(* Logix 5000 project; controller reports 1756-L63 rev 20.11; software revision 20.04; part 42 of 52 *)

        [102].log_data[71].valid := 1, [102].log_data[72].valid := 1, [102].log_data[73].valid := 1, [102].log_data[74].valid := 1, [102].log_data[75].valid := 1, [102].log_data[76].valid := 1, [102].log_data[77].valid := 1, [102].log_data[78].valid := 1, [102].log_data[79].valid := 1, [102].log_data[80].valid := 1, [102].log_data[81].valid := 1, [102].log_data[82].valid := 1, [102].log_data[83].valid := 1, [102].log_data[84].valid := 1, [102].log_data[85].valid := 1, [102].log_data[86].valid := 1, [102].log_data[87].valid := 1, [102].log_data[88].valid := 1, [102].log_data[89].valid := 1, [102].log_data[90].valid := 1, [102].log_data[91].valid := 1, [102].log_data[92].valid := 1, [102].log_data[93].valid := 1, [102].log_data[94].valid := 1, [102].log_data[95].valid := 1, [102].log_data[96].valid := 1, [102].log_data[97].valid := 1, [102].log_data[98].valid := 1, [102].log_data[99].valid := 1, [102].log_data[100].valid := 1, [102].log_data[101].valid := 1, [102].log_data[102].valid := 1, [102].log_data[103].valid := 1, [102].log_data[104].valid := 1, [102].log_data[105].valid := 1, [102].log_data[106].valid := 1, [102].log_data[107].valid := 1, [102].log_data[108].valid := 1, [102].log_data[109].valid := 1, [102].log_data[110].valid := 1, [102].log_data[111].valid := 1, [102].log_data[112].valid := 1, [102].log_data[113].valid := 1, [102].log_data[114].valid := 1, [102].log_data[115].valid := 1, [102].log_data[116].valid := 1, [102].log_data[117].valid := 1, [102].log_data[118].valid := 1, [102].log_data[119].valid := 1, [102].log_data[120].valid := 1, [102].log_data[121].valid := 1, [102].log_data[122].valid := 1, [102].log_data[123].valid := 1, [102].log_data[124].valid := 1, [102].time.Year := 2023, [102].time.Month := 1, [102].time.Day := 17, [102].time.Hour := 9, [102].time.Minute := 59, [102].time.Second := 59,
        [103].log_data[0].min := 1.0, [103].log_data[0].max := 1.0, [103].log_data[0].total := 3600.0, [103].log_data[0].time := 3600.0, [103].log_data[0].valid := 1, [103].log_data[1].max := 1.0, [103].log_data[1].total := 558.0, [103].log_data[1].time := 3600.0, [103].log_data[1].maxminute := 47, [103].log_data[1].valid := 1, [103].log_data[2].max := 1.0, [103].log_data[2].total := 554.5, [103].log_data[2].time := 3600.0, [103].log_data[2].maxminute := 47, [103].log_data[2].valid := 1, [103].log_data[3].time := 3600.0, [103].log_data[3].valid := 1, [103].log_data[4].time := 3600.0, [103].log_data[4].valid := 1, [103].log_data[5].max := 1.0, [103].log_data[5].total := 240.0, [103].log_data[5].time := 3600.0, [103].log_data[5].maxminute := 50, [103].log_data[5].valid := 1, [103].log_data[6].time := 3600.0, [103].log_data[6].valid := 1, [103].log_data[7].time := 3600.0, [103].log_data[7].valid := 1, [103].log_data[8].min := 1.0, [103].log_data[8].max := 1.0, [103].log_data[8].total := 3600.0, [103].log_data[8].time := 3600.0, [103].log_data[8].valid := 1, [103].log_data[9].min := 1.0, [103].log_data[9].max := 1.0, [103].log_data[9].total := 3600.0, [103].log_data[9].time := 3600.0, [103].log_data[9].valid := 1, [103].log_data[10].min := 1.0, [103].log_data[10].max := 1.0, [103].log_data[10].total := 3600.0, [103].log_data[10].time := 3600.0, [103].log_data[10].valid := 1, [103].log_data[11].time := 3600.0, [103].log_data[11].valid := 1, [103].log_data[12].min := 1.0, [103].log_data[12].max := 1.0, [103].log_data[12].total := 3600.0, [103].log_data[12].time := 3600.0, [103].log_data[12].valid := 1, [103].log_data[13].min := 1.0, [103].log_data[13].max := 1.0, [103].log_data[13].total := 3600.0, [103].log_data[13].time := 3600.0, [103].log_data[13].valid := 1, [103].log_data[14].time := 3600.0, [103].log_data[14].valid := 1, [103].log_data[15].time := 3600.0, [103].log_data[15].valid := 1, [103].log_data[16].time := 3600.0,
        [103].log_data[16].valid := 1, [103].log_data[17].min := 1.0, [103].log_data[17].max := 1.0, [103].log_data[17].total := 3600.0, [103].log_data[17].time := 3600.0, [103].log_data[17].valid := 1, [103].log_data[18].time := 3600.0, [103].log_data[18].valid := 1, [103].log_data[19].time := 3600.0, [103].log_data[19].valid := 1, [103].log_data[20].time := 3600.0, [103].log_data[20].valid := 1, [103].log_data[21].min := 1.0, [103].log_data[21].max := 1.0, [103].log_data[21].total := 3600.0, [103].log_data[21].time := 3600.0, [103].log_data[21].valid := 1, [103].log_data[22].time := 3600.0, [103].log_data[22].valid := 1, [103].log_data[23].time := 3600.0, [103].log_data[23].valid := 1, [103].log_data[24].time := 3600.0, [103].log_data[24].valid := 1, [103].log_data[25].time := 3600.0, [103].log_data[25].valid := 1, [103].log_data[26].time := 3600.0, [103].log_data[26].valid := 1, [103].log_data[27].time := 3600.0, [103].log_data[27].valid := 1, [103].log_data[28].time := 3600.0, [103].log_data[28].valid := 1, [103].log_data[29].min := 1.0, [103].log_data[29].max := 1.0, [103].log_data[29].total := 3600.0, [103].log_data[29].time := 3600.0, [103].log_data[29].valid := 1, [103].log_data[30].min := 1.0, [103].log_data[30].max := 1.0, [103].log_data[30].total := 3600.0, [103].log_data[30].time := 3600.0, [103].log_data[30].valid := 1, [103].log_data[31].max := 1.0, [103].log_data[31].total := 1440.7471, [103].log_data[31].time := 3600.0, [103].log_data[31].minminute := 3, [103].log_data[31].valid := 1, [103].log_data[32].max := 1.0, [103].log_data[32].total := 1629.7471, [103].log_data[32].time := 3600.0, [103].log_data[32].maxminute := 4, [103].log_data[32].valid := 1, [103].log_data[33].time := 3600.0, [103].log_data[33].valid := 1, [103].log_data[34].time := 3600.0, [103].log_data[34].valid := 1, [103].log_data[35].max := 1.0, [103].log_data[35].total := 1541.7471, [103].log_data[35].time := 3600.0, [103].log_data[35].maxminute := 10, [103].log_data[35].valid := 1,
        [103].log_data[36].max := 1.0, [103].log_data[36].total := 1616.998, [103].log_data[36].time := 3600.0, [103].log_data[36].minminute := 8, [103].log_data[36].valid := 1, [103].log_data[37].max := 7.337698, [103].log_data[37].total := 3557.1064, [103].log_data[37].time := 3600.0, [103].log_data[37].maxminute := 51, [103].log_data[37].valid := 1, [103].log_data[38].time := 3600.0, [103].log_data[38].valid := 1, [103].log_data[39].min := 0.9945885, [103].log_data[39].max := 1.0217944, [103].log_data[39].total := 3607.459, [103].log_data[39].time := 3600.0, [103].log_data[39].minminute := 6, [103].log_data[39].maxminute := 50, [103].log_data[39].valid := 1, [103].log_data[40].min := 7.5945454, [103].log_data[40].max := 7.603614, [103].log_data[40].total := 27364.693, [103].log_data[40].time := 3600.0, [103].log_data[40].minminute := 59, [103].log_data[40].maxminute := 11, [103].log_data[40].valid := 1, [103].log_data[41].min := 0.02273633, [103].log_data[41].max := 0.02411035, [103].log_data[41].total := 82.59197, [103].log_data[41].time := 3600.0, [103].log_data[41].maxminute := 16, [103].log_data[41].valid := 1, [103].log_data[42].min := 2.2916427, [103].log_data[42].max := 2.296236, [103].log_data[42].total := 8258.847, [103].log_data[42].time := 3600.0, [103].log_data[42].minminute := 6, [103].log_data[42].maxminute := 49, [103].log_data[42].valid := 1, [103].log_data[43].min := -0.27999878, [103].log_data[43].max := -0.26000214, [103].log_data[43].total := -993.9634, [103].log_data[43].time := 3600.0, [103].log_data[43].valid := 1, [103].log_data[44].min := -0.3199997, [103].log_data[44].max := -0.30000305, [103].log_data[44].total := -1080.9617, [103].log_data[44].time := 3600.0, [103].log_data[44].minminute := 2, [103].log_data[44].valid := 1, [103].log_data[45].time := 3600.0, [103].log_data[45].valid := 1, [103].log_data[46].time := 3600.0, [103].log_data[46].valid := 1, [103].log_data[47].time := 3600.0, [103].log_data[47].valid := 1, [103].log_data[48].min := 6.732198, [103].log_data[48].max := 6.899556, [103].log_data[48].total := 24363.74, [103].log_data[48].time := 3600.0,
        [103].log_data[48].minminute := 49, [103].log_data[48].maxminute := 53, [103].log_data[48].valid := 1, [103].log_data[49].min := 7.888525, [103].log_data[49].max := 9.465529, [103].log_data[49].total := 32666.957, [103].log_data[49].time := 3600.0, [103].log_data[49].maxminute := 49, [103].log_data[49].valid := 1, [103].log_data[50].min := 1.9457378, [103].log_data[50].max := 2.058684, [103].log_data[50].total := 7166.7627, [103].log_data[50].time := 3600.0, [103].log_data[50].minminute := 50, [103].log_data[50].maxminute := 58, [103].log_data[50].valid := 1, [103].log_data[51].time := 3600.0, [103].log_data[51].valid := 1, [103].log_data[52].min := -3.0800018, [103].log_data[52].max := 0.11999512, [103].log_data[52].total := -7540.314, [103].log_data[52].time := 3600.0, [103].log_data[52].minminute := 9, [103].log_data[52].maxminute := 3, [103].log_data[52].valid := 1, [103].log_data[53].min := -2.8600006, [103].log_data[53].max := 0.2599945, [103].log_data[53].total := -7208.585, [103].log_data[53].time := 3600.0, [103].log_data[53].minminute := 14, [103].log_data[53].maxminute := 30, [103].log_data[53].valid := 1, [103].log_data[54].max := 0.53, [103].log_data[54].total := 1217.2987, [103].log_data[54].time := 3600.0, [103].log_data[54].minminute := 3, [103].log_data[54].maxminute := 25, [103].log_data[54].valid := 1, [103].log_data[55].max := 0.52349997, [103].log_data[55].total := 1254.156, [103].log_data[55].time := 3600.0, [103].log_data[55].minminute := 8, [103].log_data[55].maxminute := 31, [103].log_data[55].valid := 1, [103].log_data[56].min := 0.1594997, [103].log_data[56].max := 0.16012783, [103].log_data[56].total := 575.3569, [103].log_data[56].time := 3600.0, [103].log_data[56].minminute := 39, [103].log_data[56].maxminute := 10, [103].log_data[56].valid := 1, [103].log_data[57].min := 0.23228458, [103].log_data[57].max := 0.23275566, [103].log_data[57].total := 836.9818, [103].log_data[57].time := 3600.0, [103].log_data[57].minminute := 52, [103].log_data[57].maxminute := 25, [103].log_data[57].valid := 1, [103].log_data[58].time := 3600.0, [103].log_data[58].valid := 1,
        [103].log_data[59].time := 3600.0, [103].log_data[59].valid := 1, [103].log_data[60].valid := 1, [103].log_data[61].valid := 1, [103].log_data[62].valid := 1, [103].log_data[63].valid := 1, [103].log_data[64].valid := 1, [103].log_data[65].valid := 1, [103].log_data[66].valid := 1, [103].log_data[67].valid := 1, [103].log_data[68].valid := 1, [103].log_data[69].valid := 1, [103].log_data[70].valid := 1, [103].log_data[71].valid := 1, [103].log_data[72].valid := 1, [103].log_data[73].valid := 1, [103].log_data[74].valid := 1, [103].log_data[75].valid := 1, [103].log_data[76].valid := 1, [103].log_data[77].valid := 1, [103].log_data[78].valid := 1, [103].log_data[79].valid := 1, [103].log_data[80].valid := 1, [103].log_data[81].valid := 1, [103].log_data[82].valid := 1, [103].log_data[83].valid := 1, [103].log_data[84].valid := 1, [103].log_data[85].valid := 1, [103].log_data[86].valid := 1, [103].log_data[87].valid := 1, [103].log_data[88].valid := 1, [103].log_data[89].valid := 1, [103].log_data[90].valid := 1, [103].log_data[91].valid := 1, [103].log_data[92].valid := 1, [103].log_data[93].valid := 1, [103].log_data[94].valid := 1, [103].log_data[95].valid := 1, [103].log_data[96].valid := 1, [103].log_data[97].valid := 1, [103].log_data[98].valid := 1, [103].log_data[99].valid := 1, [103].log_data[100].valid := 1, [103].log_data[101].valid := 1, [103].log_data[102].valid := 1, [103].log_data[103].valid := 1, [103].log_data[104].valid := 1, [103].log_data[105].valid := 1, [103].log_data[106].valid := 1, [103].log_data[107].valid := 1, [103].log_data[108].valid := 1, [103].log_data[109].valid := 1, [103].log_data[110].valid := 1, [103].log_data[111].valid := 1, [103].log_data[112].valid := 1, [103].log_data[113].valid := 1, [103].log_data[114].valid := 1, [103].log_data[115].valid := 1, [103].log_data[116].valid := 1, [103].log_data[117].valid := 1,
        [103].log_data[118].valid := 1, [103].log_data[119].valid := 1, [103].log_data[120].valid := 1, [103].log_data[121].valid := 1, [103].log_data[122].valid := 1, [103].log_data[123].valid := 1, [103].log_data[124].valid := 1, [103].time.Year := 2023, [103].time.Month := 1, [103].time.Day := 17, [103].time.Hour := 10, [103].time.Minute := 59, [103].time.Second := 59, [104].log_data[0].min := 1.0, [104].log_data[0].max := 1.0, [104].log_data[0].total := 3600.0, [104].log_data[0].time := 3600.0, [104].log_data[0].valid := 1, [104].log_data[1].max := 1.0, [104].log_data[1].total := 90.0, [104].log_data[1].time := 3600.0, [104].log_data[1].maxminute := 5, [104].log_data[1].valid := 1, [104].log_data[2].max := 1.0, [104].log_data[2].total := 86.5, [104].log_data[2].time := 3600.0, [104].log_data[2].maxminute := 5, [104].log_data[2].valid := 1, [104].log_data[3].time := 3600.0, [104].log_data[3].valid := 1, [104].log_data[4].time := 3600.0, [104].log_data[4].valid := 1, [104].log_data[5].time := 3600.0, [104].log_data[5].valid := 1, [104].log_data[6].time := 3600.0, [104].log_data[6].valid := 1, [104].log_data[7].time := 3600.0, [104].log_data[7].valid := 1, [104].log_data[8].min := 1.0, [104].log_data[8].max := 1.0, [104].log_data[8].total := 3600.0, [104].log_data[8].time := 3600.0, [104].log_data[8].valid := 1, [104].log_data[9].min := 1.0, [104].log_data[9].max := 1.0, [104].log_data[9].total := 3600.0, [104].log_data[9].time := 3600.0, [104].log_data[9].valid := 1, [104].log_data[10].min := 1.0, [104].log_data[10].max := 1.0, [104].log_data[10].total := 3600.0, [104].log_data[10].time := 3600.0, [104].log_data[10].valid := 1, [104].log_data[11].time := 3600.0, [104].log_data[11].valid := 1, [104].log_data[12].min := 1.0, [104].log_data[12].max := 1.0, [104].log_data[12].total := 3600.0, [104].log_data[12].time := 3600.0, [104].log_data[12].valid := 1,
        [104].log_data[13].min := 1.0, [104].log_data[13].max := 1.0, [104].log_data[13].total := 3600.0, [104].log_data[13].time := 3600.0, [104].log_data[13].valid := 1, [104].log_data[14].time := 3600.0, [104].log_data[14].valid := 1, [104].log_data[15].time := 3600.0, [104].log_data[15].valid := 1, [104].log_data[16].time := 3600.0, [104].log_data[16].valid := 1, [104].log_data[17].min := 1.0, [104].log_data[17].max := 1.0, [104].log_data[17].total := 3600.0, [104].log_data[17].time := 3600.0, [104].log_data[17].valid := 1, [104].log_data[18].time := 3600.0, [104].log_data[18].valid := 1, [104].log_data[19].time := 3600.0, [104].log_data[19].valid := 1, [104].log_data[20].time := 3600.0, [104].log_data[20].valid := 1, [104].log_data[21].min := 1.0, [104].log_data[21].max := 1.0, [104].log_data[21].total := 3600.0, [104].log_data[21].time := 3600.0, [104].log_data[21].valid := 1, [104].log_data[22].time := 3600.0, [104].log_data[22].valid := 1, [104].log_data[23].time := 3600.0, [104].log_data[23].valid := 1, [104].log_data[24].time := 3600.0, [104].log_data[24].valid := 1, [104].log_data[25].time := 3600.0, [104].log_data[25].valid := 1, [104].log_data[26].time := 3600.0, [104].log_data[26].valid := 1, [104].log_data[27].time := 3600.0, [104].log_data[27].valid := 1, [104].log_data[28].time := 3600.0, [104].log_data[28].valid := 1, [104].log_data[29].min := 1.0, [104].log_data[29].max := 1.0, [104].log_data[29].total := 3600.0, [104].log_data[29].time := 3600.0, [104].log_data[29].valid := 1, [104].log_data[30].min := 1.0, [104].log_data[30].max := 1.0, [104].log_data[30].total := 3600.0, [104].log_data[30].time := 3600.0, [104].log_data[30].valid := 1, [104].log_data[31].max := 1.0, [104].log_data[31].total := 1469.498, [104].log_data[31].time := 3600.0, [104].log_data[31].minminute := 6, [104].log_data[31].valid := 1, [104].log_data[32].max := 1.0, [104].log_data[32].total := 1629.998, [104].log_data[32].time := 3600.0, [104].log_data[32].maxminute := 7,
        [104].log_data[32].valid := 1, [104].log_data[33].time := 3600.0, [104].log_data[33].valid := 1, [104].log_data[34].time := 3600.0, [104].log_data[34].valid := 1, [104].log_data[35].max := 1.0, [104].log_data[35].total := 1440.498, [104].log_data[35].time := 3600.0, [104].log_data[35].minminute := 1, [104].log_data[35].valid := 1, [104].log_data[36].max := 1.0, [104].log_data[36].total := 1629.7471, [104].log_data[36].time := 3600.0, [104].log_data[36].maxminute := 2, [104].log_data[36].valid := 1, [104].log_data[37].max := 2.600009, [104].log_data[37].total := 99.13652, [104].log_data[37].time := 3600.0, [104].log_data[37].maxminute := 5, [104].log_data[37].valid := 1, [104].log_data[38].time := 3600.0, [104].log_data[38].valid := 1, [104].log_data[39].min := 0.9957663, [104].log_data[39].max := 1.0073081, [104].log_data[39].total := 3607.94, [104].log_data[39].time := 3600.0, [104].log_data[39].minminute := 4, [104].log_data[39].maxminute := 43, [104].log_data[39].valid := 1, [104].log_data[40].min := 7.5802555, [104].log_data[40].max := 7.6093855, [104].log_data[40].total := 27364.307, [104].log_data[40].time := 3600.0, [104].log_data[40].minminute := 45, [104].log_data[40].maxminute := 48, [104].log_data[40].valid := 1, [104].log_data[41].min := 0.02273633, [104].log_data[41].max := 0.023128908, [104].log_data[41].total := 82.71829, [104].log_data[41].time := 3600.0, [104].log_data[41].valid := 1, [104].log_data[42].min := 2.2911716, [104].log_data[42].max := 2.296118, [104].log_data[42].total := 8258.796, [104].log_data[42].time := 3600.0, [104].log_data[42].minminute := 24, [104].log_data[42].maxminute := 29, [104].log_data[42].valid := 1, [104].log_data[43].min := -0.27999878, [104].log_data[43].max := -0.26000214, [104].log_data[43].total := -1007.0374, [104].log_data[43].time := 3600.0, [104].log_data[43].valid := 1, [104].log_data[44].min := -0.3199997, [104].log_data[44].max := -0.30000305, [104].log_data[44].total := -1100.4613, [104].log_data[44].time := 3600.0, [104].log_data[44].valid := 1, [104].log_data[45].time := 3600.0, [104].log_data[45].valid := 1,
        [104].log_data[46].time := 3600.0, [104].log_data[46].valid := 1, [104].log_data[47].time := 3600.0, [104].log_data[47].valid := 1, [104].log_data[48].min := 6.578031, [104].log_data[48].max := 6.801175, [104].log_data[48].total := 24174.486, [104].log_data[48].time := 3600.0, [104].log_data[48].minminute := 16, [104].log_data[48].maxminute := 33, [104].log_data[48].valid := 1, [104].log_data[49].min := 6.728443, [104].log_data[49].max := 9.348344, [104].log_data[49].total := 28856.195, [104].log_data[49].time := 3600.0, [104].log_data[49].minminute := 18, [104].log_data[49].maxminute := 59, [104].log_data[49].valid := 1, [104].log_data[50].min := 1.9717662, [104].log_data[50].max := 2.0559752, [104].log_data[50].total := 7259.038, [104].log_data[50].time := 3600.0, [104].log_data[50].minminute := 59, [104].log_data[50].maxminute := 1, [104].log_data[50].valid := 1, [104].log_data[51].time := 3600.0, [104].log_data[51].valid := 1, [104].log_data[52].min := -2.880005, [104].log_data[52].max := 0.11999512, [104].log_data[52].total := -7743.9883, [104].log_data[52].time := 3600.0, [104].log_data[52].minminute := 7, [104].log_data[52].maxminute := 6, [104].log_data[52].valid := 1, [104].log_data[53].min := -2.540001, [104].log_data[53].max := 0.2400055, [104].log_data[53].total := -7001.7065, [104].log_data[53].time := 3600.0, [104].log_data[53].minminute := 55, [104].log_data[53].maxminute := 2, [104].log_data[53].valid := 1, [104].log_data[54].max := 0.5215, [104].log_data[54].total := 1230.9836, [104].log_data[54].time := 3600.0, [104].log_data[54].minminute := 6, [104].log_data[54].maxminute := 18, [104].log_data[54].valid := 1, [104].log_data[55].max := 0.52099997, [104].log_data[55].total := 1217.138, [104].log_data[55].time := 3600.0, [104].log_data[55].minminute := 1, [104].log_data[55].maxminute := 55, [104].log_data[55].valid := 1, [104].log_data[56].min := 0.15957822, [104].log_data[56].max := 0.16001005, [104].log_data[56].total := 575.15814, [104].log_data[56].time := 3600.0, [104].log_data[56].minminute := 15, [104].log_data[56].maxminute := 7, [104].log_data[56].valid := 1,
        [104].log_data[57].min := 0.2303609, [104].log_data[57].max := 0.23267715, [104].log_data[57].total := 832.2318, [104].log_data[57].time := 3600.0, [104].log_data[57].minminute := 37, [104].log_data[57].valid := 1, [104].log_data[58].time := 3600.0, [104].log_data[58].valid := 1, [104].log_data[59].time := 3600.0, [104].log_data[59].valid := 1, [104].log_data[60].valid := 1, [104].log_data[61].valid := 1, [104].log_data[62].valid := 1, [104].log_data[63].valid := 1, [104].log_data[64].valid := 1, [104].log_data[65].valid := 1, [104].log_data[66].valid := 1, [104].log_data[67].valid := 1, [104].log_data[68].valid := 1, [104].log_data[69].valid := 1, [104].log_data[70].valid := 1, [104].log_data[71].valid := 1, [104].log_data[72].valid := 1, [104].log_data[73].valid := 1, [104].log_data[74].valid := 1, [104].log_data[75].valid := 1, [104].log_data[76].valid := 1, [104].log_data[77].valid := 1, [104].log_data[78].valid := 1, [104].log_data[79].valid := 1, [104].log_data[80].valid := 1, [104].log_data[81].valid := 1, [104].log_data[82].valid := 1, [104].log_data[83].valid := 1, [104].log_data[84].valid := 1, [104].log_data[85].valid := 1, [104].log_data[86].valid := 1, [104].log_data[87].valid := 1, [104].log_data[88].valid := 1, [104].log_data[89].valid := 1, [104].log_data[90].valid := 1, [104].log_data[91].valid := 1, [104].log_data[92].valid := 1, [104].log_data[93].valid := 1, [104].log_data[94].valid := 1, [104].log_data[95].valid := 1, [104].log_data[96].valid := 1, [104].log_data[97].valid := 1, [104].log_data[98].valid := 1, [104].log_data[99].valid := 1, [104].log_data[100].valid := 1, [104].log_data[101].valid := 1, [104].log_data[102].valid := 1, [104].log_data[103].valid := 1, [104].log_data[104].valid := 1, [104].log_data[105].valid := 1, [104].log_data[106].valid := 1, [104].log_data[107].valid := 1, [104].log_data[108].valid := 1, [104].log_data[109].valid := 1,
        [104].log_data[110].valid := 1, [104].log_data[111].valid := 1, [104].log_data[112].valid := 1, [104].log_data[113].valid := 1, [104].log_data[114].valid := 1, [104].log_data[115].valid := 1, [104].log_data[116].valid := 1, [104].log_data[117].valid := 1, [104].log_data[118].valid := 1, [104].log_data[119].valid := 1, [104].log_data[120].valid := 1, [104].log_data[121].valid := 1, [104].log_data[122].valid := 1, [104].log_data[123].valid := 1, [104].log_data[124].valid := 1, [104].time.Year := 2023, [104].time.Month := 1, [104].time.Day := 17, [104].time.Hour := 11, [104].time.Minute := 59, [104].time.Second := 59, [105].log_data[0].min := 1.0, [105].log_data[0].max := 1.0, [105].log_data[0].total := 3600.0, [105].log_data[0].time := 3600.0, [105].log_data[0].valid := 1, [105].log_data[1].max := 1.0, [105].log_data[1].total := 544.0, [105].log_data[1].time := 3600.0, [105].log_data[1].maxminute := 21, [105].log_data[1].valid := 1, [105].log_data[2].max := 1.0, [105].log_data[2].total := 540.5, [105].log_data[2].time := 3600.0, [105].log_data[2].maxminute := 21, [105].log_data[2].valid := 1, [105].log_data[3].time := 3600.0, [105].log_data[3].valid := 1, [105].log_data[4].time := 3600.0, [105].log_data[4].valid := 1, [105].log_data[5].max := 1.0, [105].log_data[5].total := 245.0, [105].log_data[5].time := 3600.0, [105].log_data[5].maxminute := 23, [105].log_data[5].valid := 1, [105].log_data[6].time := 3600.0, [105].log_data[6].valid := 1, [105].log_data[7].time := 3600.0, [105].log_data[7].valid := 1, [105].log_data[8].min := 1.0, [105].log_data[8].max := 1.0, [105].log_data[8].total := 3600.0, [105].log_data[8].time := 3600.0, [105].log_data[8].valid := 1, [105].log_data[9].min := 1.0, [105].log_data[9].max := 1.0, [105].log_data[9].total := 3600.0, [105].log_data[9].time := 3600.0, [105].log_data[9].valid := 1, [105].log_data[10].min := 1.0,
        [105].log_data[10].max := 1.0, [105].log_data[10].total := 3600.0, [105].log_data[10].time := 3600.0, [105].log_data[10].valid := 1, [105].log_data[11].time := 3600.0, [105].log_data[11].valid := 1, [105].log_data[12].min := 1.0, [105].log_data[12].max := 1.0, [105].log_data[12].total := 3600.0, [105].log_data[12].time := 3600.0, [105].log_data[12].valid := 1, [105].log_data[13].min := 1.0, [105].log_data[13].max := 1.0, [105].log_data[13].total := 3600.0, [105].log_data[13].time := 3600.0, [105].log_data[13].valid := 1, [105].log_data[14].time := 3600.0, [105].log_data[14].valid := 1, [105].log_data[15].time := 3600.0, [105].log_data[15].valid := 1, [105].log_data[16].time := 3600.0, [105].log_data[16].valid := 1, [105].log_data[17].min := 1.0, [105].log_data[17].max := 1.0, [105].log_data[17].total := 3600.0, [105].log_data[17].time := 3600.0, [105].log_data[17].valid := 1, [105].log_data[18].time := 3600.0, [105].log_data[18].valid := 1, [105].log_data[19].time := 3600.0, [105].log_data[19].valid := 1, [105].log_data[20].time := 3600.0, [105].log_data[20].valid := 1, [105].log_data[21].min := 1.0, [105].log_data[21].max := 1.0, [105].log_data[21].total := 3600.0, [105].log_data[21].time := 3600.0, [105].log_data[21].valid := 1, [105].log_data[22].time := 3600.0, [105].log_data[22].valid := 1, [105].log_data[23].time := 3600.0, [105].log_data[23].valid := 1, [105].log_data[24].time := 3600.0, [105].log_data[24].valid := 1, [105].log_data[25].time := 3600.0, [105].log_data[25].valid := 1, [105].log_data[26].time := 3600.0, [105].log_data[26].valid := 1, [105].log_data[27].time := 3600.0, [105].log_data[27].valid := 1, [105].log_data[28].time := 3600.0, [105].log_data[28].valid := 1, [105].log_data[29].min := 1.0, [105].log_data[29].max := 1.0, [105].log_data[29].total := 3600.0, [105].log_data[29].time := 3600.0, [105].log_data[29].valid := 1, [105].log_data[30].min := 1.0, [105].log_data[30].max := 1.0, [105].log_data[30].total := 3600.0,
        [105].log_data[30].time := 3600.0, [105].log_data[30].valid := 1, [105].log_data[31].max := 1.0, [105].log_data[31].total := 1629.998, [105].log_data[31].time := 3600.0, [105].log_data[31].valid := 1, [105].log_data[32].max := 1.0, [105].log_data[32].total := 1500.2471, [105].log_data[32].time := 3600.0, [105].log_data[32].maxminute := 11, [105].log_data[32].valid := 1, [105].log_data[33].time := 3600.0, [105].log_data[33].valid := 1, [105].log_data[34].time := 3600.0, [105].log_data[34].valid := 1, [105].log_data[35].max := 1.0, [105].log_data[35].total := 1440.7471, [105].log_data[35].time := 3600.0, [105].log_data[35].minminute := 4, [105].log_data[35].valid := 1, [105].log_data[36].max := 1.0, [105].log_data[36].total := 1629.998, [105].log_data[36].time := 3600.0, [105].log_data[36].maxminute := 6, [105].log_data[36].valid := 1, [105].log_data[37].max := 7.473924, [105].log_data[37].total := 3521.814, [105].log_data[37].time := 3600.0, [105].log_data[37].maxminute := 23, [105].log_data[37].valid := 1, [105].log_data[38].time := 3600.0, [105].log_data[38].valid := 1, [105].log_data[39].min := 0.9950596, [105].log_data[39].max := 1.0221478, [105].log_data[39].total := 3609.72, [105].log_data[39].time := 3600.0, [105].log_data[39].minminute := 39, [105].log_data[39].maxminute := 28, [105].log_data[39].valid := 1, [105].log_data[40].min := 7.5928965, [105].log_data[40].max := 7.6077366, [105].log_data[40].total := 27365.082, [105].log_data[40].time := 3600.0, [105].log_data[40].minminute := 52, [105].log_data[40].maxminute := 54, [105].log_data[40].valid := 1, [105].log_data[41].min := 0.02273633, [105].log_data[41].max := 0.023325196, [105].log_data[41].total := 82.87387, [105].log_data[41].time := 3600.0, [105].log_data[41].minminute := 3, [105].log_data[41].maxminute := 20, [105].log_data[41].valid := 1, [105].log_data[42].min := 2.2917604, [105].log_data[42].max := 2.2964714, [105].log_data[42].total := 8259.048, [105].log_data[42].time := 3600.0, [105].log_data[42].minminute := 22, [105].log_data[42].maxminute := 4, [105].log_data[42].valid := 1,
        [105].log_data[43].min := -0.27999878, [105].log_data[43].max := -0.26000214, [105].log_data[43].total := -998.42554, [105].log_data[43].time := 3600.0, [105].log_data[43].valid := 1, [105].log_data[44].min := -0.3199997, [105].log_data[44].max := -0.30000305, [105].log_data[44].total := -1085.1592, [105].log_data[44].time := 3600.0, [105].log_data[44].valid := 1, [105].log_data[45].time := 3600.0, [105].log_data[45].valid := 1, [105].log_data[46].time := 3600.0, [105].log_data[46].valid := 1, [105].log_data[47].time := 3600.0, [105].log_data[47].valid := 1, [105].log_data[48].min := 6.5708866, [105].log_data[48].max := 6.909449, [105].log_data[48].total := 24175.59, [105].log_data[48].time := 3600.0, [105].log_data[48].minminute := 52, [105].log_data[48].maxminute := 26, [105].log_data[48].valid := 1, [105].log_data[49].min := 6.671519, [105].log_data[49].max := 9.436871, [105].log_data[49].total := 29516.545, [105].log_data[49].time := 3600.0, [105].log_data[49].minminute := 47, [105].log_data[49].maxminute := 17, [105].log_data[49].valid := 1, [105].log_data[50].min := 1.9406737, [105].log_data[50].max := 2.0525599, [105].log_data[50].total := 7204.415, [105].log_data[50].time := 3600.0, [105].log_data[50].minminute := 23, [105].log_data[50].maxminute := 31, [105].log_data[50].valid := 1, [105].log_data[51].time := 3600.0, [105].log_data[51].valid := 1, [105].log_data[52].min := -2.9400024, [105].log_data[52].max := 0.11999512, [105].log_data[52].total := -7841.4717, [105].log_data[52].time := 3600.0, [105].log_data[52].minminute := 32, [105].log_data[52].valid := 1, [105].log_data[53].min := -2.4800034, [105].log_data[53].max := 0.22000122, [105].log_data[53].total := -7097.0947, [105].log_data[53].time := 3600.0, [105].log_data[53].minminute := 25, [105].log_data[53].maxminute := 37, [105].log_data[53].valid := 1, [105].log_data[54].max := 0.5475, [105].log_data[54].total := 1241.1823, [105].log_data[54].time := 3600.0, [105].log_data[54].maxminute := 11, [105].log_data[54].valid := 1, [105].log_data[55].max := 0.52349997, [105].log_data[55].total := 1217.1405, [105].log_data[55].time := 3600.0,
        [105].log_data[55].minminute := 4, [105].log_data[55].maxminute := 16, [105].log_data[55].valid := 1, [105].log_data[56].min := 0.15957822, [105].log_data[56].max := 0.16001005, [105].log_data[56].total := 575.1107, [105].log_data[56].time := 3600.0, [105].log_data[56].minminute := 42, [105].log_data[56].maxminute := 2, [105].log_data[56].valid := 1, [105].log_data[57].min := 0.22894761, [105].log_data[57].max := 0.23083198, [105].log_data[57].total := 829.5313, [105].log_data[57].time := 3600.0, [105].log_data[57].minminute := 59, [105].log_data[57].maxminute := 15, [105].log_data[57].valid := 1, [105].log_data[58].time := 3600.0, [105].log_data[58].valid := 1, [105].log_data[59].time := 3600.0, [105].log_data[59].valid := 1, [105].log_data[60].valid := 1, [105].log_data[61].valid := 1, [105].log_data[62].valid := 1, [105].log_data[63].valid := 1, [105].log_data[64].valid := 1, [105].log_data[65].valid := 1, [105].log_data[66].valid := 1, [105].log_data[67].valid := 1, [105].log_data[68].valid := 1, [105].log_data[69].valid := 1, [105].log_data[70].valid := 1, [105].log_data[71].valid := 1, [105].log_data[72].valid := 1, [105].log_data[73].valid := 1, [105].log_data[74].valid := 1, [105].log_data[75].valid := 1, [105].log_data[76].valid := 1, [105].log_data[77].valid := 1, [105].log_data[78].valid := 1, [105].log_data[79].valid := 1, [105].log_data[80].valid := 1, [105].log_data[81].valid := 1, [105].log_data[82].valid := 1, [105].log_data[83].valid := 1, [105].log_data[84].valid := 1, [105].log_data[85].valid := 1, [105].log_data[86].valid := 1, [105].log_data[87].valid := 1, [105].log_data[88].valid := 1, [105].log_data[89].valid := 1, [105].log_data[90].valid := 1, [105].log_data[91].valid := 1, [105].log_data[92].valid := 1, [105].log_data[93].valid := 1, [105].log_data[94].valid := 1, [105].log_data[95].valid := 1, [105].log_data[96].valid := 1, [105].log_data[97].valid := 1, [105].log_data[98].valid := 1,
        [105].log_data[99].valid := 1, [105].log_data[100].valid := 1, [105].log_data[101].valid := 1, [105].log_data[102].valid := 1, [105].log_data[103].valid := 1, [105].log_data[104].valid := 1, [105].log_data[105].valid := 1, [105].log_data[106].valid := 1, [105].log_data[107].valid := 1, [105].log_data[108].valid := 1, [105].log_data[109].valid := 1, [105].log_data[110].valid := 1, [105].log_data[111].valid := 1, [105].log_data[112].valid := 1, [105].log_data[113].valid := 1, [105].log_data[114].valid := 1, [105].log_data[115].valid := 1, [105].log_data[116].valid := 1, [105].log_data[117].valid := 1, [105].log_data[118].valid := 1, [105].log_data[119].valid := 1, [105].log_data[120].valid := 1, [105].log_data[121].valid := 1, [105].log_data[122].valid := 1, [105].log_data[123].valid := 1, [105].log_data[124].valid := 1, [105].time.Year := 2023, [105].time.Month := 1, [105].time.Day := 17, [105].time.Hour := 12, [105].time.Minute := 59, [105].time.Second := 59, [106].log_data[0].min := 1.0, [106].log_data[0].max := 1.0, [106].log_data[0].total := 3600.0, [106].log_data[0].time := 3600.0, [106].log_data[0].valid := 1, [106].log_data[1].time := 3600.0, [106].log_data[1].valid := 1, [106].log_data[2].time := 3600.0, [106].log_data[2].valid := 1, [106].log_data[3].time := 3600.0, [106].log_data[3].valid := 1, [106].log_data[4].time := 3600.0, [106].log_data[4].valid := 1, [106].log_data[5].time := 3600.0, [106].log_data[5].valid := 1, [106].log_data[6].time := 3600.0, [106].log_data[6].valid := 1, [106].log_data[7].time := 3600.0, [106].log_data[7].valid := 1, [106].log_data[8].min := 1.0, [106].log_data[8].max := 1.0, [106].log_data[8].total := 3600.0, [106].log_data[8].time := 3600.0, [106].log_data[8].valid := 1, [106].log_data[9].min := 1.0, [106].log_data[9].max := 1.0, [106].log_data[9].total := 3600.0, [106].log_data[9].time := 3600.0,
        [106].log_data[9].valid := 1, [106].log_data[10].min := 1.0, [106].log_data[10].max := 1.0, [106].log_data[10].total := 3600.0, [106].log_data[10].time := 3600.0, [106].log_data[10].valid := 1, [106].log_data[11].time := 3600.0, [106].log_data[11].valid := 1, [106].log_data[12].min := 1.0, [106].log_data[12].max := 1.0, [106].log_data[12].total := 3600.0, [106].log_data[12].time := 3600.0, [106].log_data[12].valid := 1, [106].log_data[13].min := 1.0, [106].log_data[13].max := 1.0, [106].log_data[13].total := 3600.0, [106].log_data[13].time := 3600.0, [106].log_data[13].valid := 1, [106].log_data[14].time := 3600.0, [106].log_data[14].valid := 1, [106].log_data[15].time := 3600.0, [106].log_data[15].valid := 1, [106].log_data[16].time := 3600.0, [106].log_data[16].valid := 1, [106].log_data[17].min := 1.0, [106].log_data[17].max := 1.0, [106].log_data[17].total := 3600.0, [106].log_data[17].time := 3600.0, [106].log_data[17].valid := 1, [106].log_data[18].time := 3600.0, [106].log_data[18].valid := 1, [106].log_data[19].time := 3600.0, [106].log_data[19].valid := 1, [106].log_data[20].time := 3600.0, [106].log_data[20].valid := 1, [106].log_data[21].min := 1.0, [106].log_data[21].max := 1.0, [106].log_data[21].total := 3600.0, [106].log_data[21].time := 3600.0, [106].log_data[21].valid := 1, [106].log_data[22].time := 3600.0, [106].log_data[22].valid := 1, [106].log_data[23].time := 3600.0, [106].log_data[23].valid := 1, [106].log_data[24].time := 3600.0, [106].log_data[24].valid := 1, [106].log_data[25].time := 3600.0, [106].log_data[25].valid := 1, [106].log_data[26].time := 3600.0, [106].log_data[26].valid := 1, [106].log_data[27].time := 3600.0, [106].log_data[27].valid := 1, [106].log_data[28].time := 3600.0, [106].log_data[28].valid := 1, [106].log_data[29].min := 1.0, [106].log_data[29].max := 1.0, [106].log_data[29].total := 3600.0, [106].log_data[29].time := 3600.0, [106].log_data[29].valid := 1, [106].log_data[30].min := 1.0,
        [106].log_data[30].max := 1.0, [106].log_data[30].total := 3600.0, [106].log_data[30].time := 3600.0, [106].log_data[30].valid := 1, [106].log_data[31].max := 1.0, [106].log_data[31].total := 1629.998, [106].log_data[31].time := 3600.0, [106].log_data[31].maxminute := 3, [106].log_data[31].valid := 1, [106].log_data[32].max := 1.0, [106].log_data[32].total := 1440.998, [106].log_data[32].time := 3600.0, [106].log_data[32].minminute := 2, [106].log_data[32].valid := 1, [106].log_data[33].time := 3600.0, [106].log_data[33].valid := 1, [106].log_data[34].time := 3600.0, [106].log_data[34].valid := 1, [106].log_data[35].max := 1.0, [106].log_data[35].total := 1552.498, [106].log_data[35].time := 3600.0, [106].log_data[35].minminute := 7, [106].log_data[35].valid := 1, [106].log_data[36].max := 1.0, [106].log_data[36].total := 1606.2471, [106].log_data[36].time := 3600.0, [106].log_data[36].maxminute := 9, [106].log_data[36].valid := 1, [106].log_data[37].time := 3600.0, [106].log_data[37].valid := 1, [106].log_data[38].time := 3600.0, [106].log_data[38].valid := 1, [106].log_data[39].min := 0.9951773, [106].log_data[39].max := 1.005306, [106].log_data[39].total := 3602.8955, [106].log_data[39].time := 3600.0, [106].log_data[39].minminute := 20, [106].log_data[39].maxminute := 2, [106].log_data[39].valid := 1, [106].log_data[40].min := 7.590149, [106].log_data[40].max := 7.6093855, [106].log_data[40].total := 27366.457, [106].log_data[40].time := 3600.0, [106].log_data[40].maxminute := 57, [106].log_data[40].valid := 1, [106].log_data[41].min := 0.02273633, [106].log_data[41].max := 0.023325196, [106].log_data[41].total := 82.77345, [106].log_data[41].time := 3600.0, [106].log_data[41].maxminute := 13, [106].log_data[41].valid := 1, [106].log_data[42].min := 2.2912893, [106].log_data[42].max := 2.2963536, [106].log_data[42].total := 8259.094, [106].log_data[42].time := 3600.0, [106].log_data[42].minminute := 4, [106].log_data[42].maxminute := 23, [106].log_data[42].valid := 1, [106].log_data[43].min := -0.27999878, [106].log_data[43].max := -0.26000214,
        [106].log_data[43].total := -958.63666, [106].log_data[43].time := 3600.0, [106].log_data[43].valid := 1, [106].log_data[44].min := -0.3199997, [106].log_data[44].max := -0.30000305, [106].log_data[44].total := -1080.1211, [106].log_data[44].time := 3600.0, [106].log_data[44].minminute := 14, [106].log_data[44].valid := 1, [106].log_data[45].time := 3600.0, [106].log_data[45].valid := 1, [106].log_data[46].time := 3600.0, [106].log_data[46].valid := 1, [106].log_data[47].time := 3600.0, [106].log_data[47].valid := 1, [106].log_data[48].min := 6.6893287, [106].log_data[48].max := 6.7984266, [106].log_data[48].total := 24335.342, [106].log_data[48].time := 3600.0, [106].log_data[48].maxminute := 8, [106].log_data[48].valid := 1, [106].log_data[49].min := 7.3436203, [106].log_data[49].max := 9.422739, [106].log_data[49].total := 32471.102, [106].log_data[49].time := 3600.0, [106].log_data[49].maxminute := 58, [106].log_data[49].valid := 1, [106].log_data[50].min := 1.9308983, [106].log_data[50].max := 2.0202894, [106].log_data[50].total := 7113.0415, [106].log_data[50].time := 3600.0, [106].log_data[50].minminute := 59, [106].log_data[50].valid := 1, [106].log_data[51].time := 3600.0, [106].log_data[51].valid := 1, [106].log_data[52].min := -2.9400024, [106].log_data[52].max := 0.11999512, [106].log_data[52].total := -7666.553, [106].log_data[52].time := 3600.0, [106].log_data[52].minminute := 45, [106].log_data[52].maxminute := 2, [106].log_data[52].valid := 1, [106].log_data[53].min := -2.5200043, [106].log_data[53].max := 0.19999695, [106].log_data[53].total := -7388.948, [106].log_data[53].time := 3600.0, [106].log_data[53].minminute := 5, [106].log_data[53].maxminute := 30, [106].log_data[53].valid := 1, [106].log_data[54].max := 0.525, [106].log_data[54].total := 1217.3862, [106].log_data[54].time := 3600.0, [106].log_data[54].minminute := 2, [106].log_data[54].maxminute := 56, [106].log_data[54].valid := 1, [106].log_data[55].max := 0.5195, [106].log_data[55].total := 1254.2628, [106].log_data[55].time := 3600.0, [106].log_data[55].minminute := 7, [106].log_data[55].maxminute := 19,
        [106].log_data[55].valid := 1, [106].log_data[56].min := 0.15957822, [106].log_data[56].max := 0.1599708, [106].log_data[56].total := 575.0373, [106].log_data[56].time := 3600.0, [106].log_data[56].minminute := 27, [106].log_data[56].maxminute := 6, [106].log_data[56].valid := 1, [106].log_data[57].min := 0.22882983, [106].log_data[57].max := 0.22926167, [106].log_data[57].total := 824.3691, [106].log_data[57].time := 3600.0, [106].log_data[57].maxminute := 35, [106].log_data[57].valid := 1, [106].log_data[58].time := 3600.0, [106].log_data[58].valid := 1, [106].log_data[59].time := 3600.0, [106].log_data[59].valid := 1, [106].log_data[60].valid := 1, [106].log_data[61].valid := 1, [106].log_data[62].valid := 1, [106].log_data[63].valid := 1, [106].log_data[64].valid := 1, [106].log_data[65].valid := 1, [106].log_data[66].valid := 1, [106].log_data[67].valid := 1, [106].log_data[68].valid := 1, [106].log_data[69].valid := 1, [106].log_data[70].valid := 1, [106].log_data[71].valid := 1, [106].log_data[72].valid := 1, [106].log_data[73].valid := 1, [106].log_data[74].valid := 1, [106].log_data[75].valid := 1, [106].log_data[76].valid := 1, [106].log_data[77].valid := 1, [106].log_data[78].valid := 1, [106].log_data[79].valid := 1, [106].log_data[80].valid := 1, [106].log_data[81].valid := 1, [106].log_data[82].valid := 1, [106].log_data[83].valid := 1, [106].log_data[84].valid := 1, [106].log_data[85].valid := 1, [106].log_data[86].valid := 1, [106].log_data[87].valid := 1, [106].log_data[88].valid := 1, [106].log_data[89].valid := 1, [106].log_data[90].valid := 1, [106].log_data[91].valid := 1, [106].log_data[92].valid := 1, [106].log_data[93].valid := 1, [106].log_data[94].valid := 1, [106].log_data[95].valid := 1, [106].log_data[96].valid := 1, [106].log_data[97].valid := 1, [106].log_data[98].valid := 1, [106].log_data[99].valid := 1, [106].log_data[100].valid := 1, [106].log_data[101].valid := 1,
        [106].log_data[102].valid := 1, [106].log_data[103].valid := 1, [106].log_data[104].valid := 1, [106].log_data[105].valid := 1, [106].log_data[106].valid := 1, [106].log_data[107].valid := 1, [106].log_data[108].valid := 1, [106].log_data[109].valid := 1, [106].log_data[110].valid := 1, [106].log_data[111].valid := 1, [106].log_data[112].valid := 1, [106].log_data[113].valid := 1, [106].log_data[114].valid := 1, [106].log_data[115].valid := 1, [106].log_data[116].valid := 1, [106].log_data[117].valid := 1, [106].log_data[118].valid := 1, [106].log_data[119].valid := 1, [106].log_data[120].valid := 1, [106].log_data[121].valid := 1, [106].log_data[122].valid := 1, [106].log_data[123].valid := 1, [106].log_data[124].valid := 1, [106].time.Year := 2023, [106].time.Month := 1, [106].time.Day := 17, [106].time.Hour := 13, [106].time.Minute := 59, [106].time.Second := 59, [107].log_data[0].min := 1.0, [107].log_data[0].max := 1.0, [107].log_data[0].total := 3600.0, [107].log_data[0].time := 3600.0, [107].log_data[0].valid := 1, [107].log_data[1].max := 1.0, [107].log_data[1].total := 564.0, [107].log_data[1].time := 3600.0, [107].log_data[1].maxminute := 14, [107].log_data[1].valid := 1, [107].log_data[2].max := 1.0, [107].log_data[2].total := 560.5, [107].log_data[2].time := 3600.0, [107].log_data[2].maxminute := 14, [107].log_data[2].valid := 1, [107].log_data[3].time := 3600.0, [107].log_data[3].valid := 1, [107].log_data[4].time := 3600.0, [107].log_data[4].valid := 1, [107].log_data[5].max := 1.0, [107].log_data[5].total := 238.5, [107].log_data[5].time := 3600.0, [107].log_data[5].maxminute := 17, [107].log_data[5].valid := 1, [107].log_data[6].time := 3600.0, [107].log_data[6].valid := 1, [107].log_data[7].time := 3600.0, [107].log_data[7].valid := 1, [107].log_data[8].min := 1.0, [107].log_data[8].max := 1.0, [107].log_data[8].total := 3600.0,
        [107].log_data[8].time := 3600.0, [107].log_data[8].valid := 1, [107].log_data[9].min := 1.0, [107].log_data[9].max := 1.0, [107].log_data[9].total := 3600.0, [107].log_data[9].time := 3600.0, [107].log_data[9].valid := 1, [107].log_data[10].min := 1.0, [107].log_data[10].max := 1.0, [107].log_data[10].total := 3600.0, [107].log_data[10].time := 3600.0, [107].log_data[10].valid := 1, [107].log_data[11].time := 3600.0, [107].log_data[11].valid := 1, [107].log_data[12].min := 1.0, [107].log_data[12].max := 1.0, [107].log_data[12].total := 3600.0, [107].log_data[12].time := 3600.0, [107].log_data[12].valid := 1, [107].log_data[13].min := 1.0, [107].log_data[13].max := 1.0, [107].log_data[13].total := 3600.0, [107].log_data[13].time := 3600.0, [107].log_data[13].valid := 1, [107].log_data[14].time := 3600.0, [107].log_data[14].valid := 1, [107].log_data[15].time := 3600.0, [107].log_data[15].valid := 1, [107].log_data[16].time := 3600.0, [107].log_data[16].valid := 1, [107].log_data[17].min := 1.0, [107].log_data[17].max := 1.0, [107].log_data[17].total := 3600.0, [107].log_data[17].time := 3600.0, [107].log_data[17].valid := 1, [107].log_data[18].time := 3600.0, [107].log_data[18].valid := 1, [107].log_data[19].time := 3600.0, [107].log_data[19].valid := 1, [107].log_data[20].time := 3600.0, [107].log_data[20].valid := 1, [107].log_data[21].min := 1.0, [107].log_data[21].max := 1.0, [107].log_data[21].total := 3600.0, [107].log_data[21].time := 3600.0, [107].log_data[21].valid := 1, [107].log_data[22].time := 3600.0, [107].log_data[22].valid := 1, [107].log_data[23].time := 3600.0, [107].log_data[23].valid := 1, [107].log_data[24].time := 3600.0, [107].log_data[24].valid := 1, [107].log_data[25].time := 3600.0, [107].log_data[25].valid := 1, [107].log_data[26].time := 3600.0, [107].log_data[26].valid := 1, [107].log_data[27].time := 3600.0, [107].log_data[27].valid := 1, [107].log_data[28].time := 3600.0, [107].log_data[28].valid := 1,
        [107].log_data[29].min := 1.0, [107].log_data[29].max := 1.0, [107].log_data[29].total := 3600.0, [107].log_data[29].time := 3600.0, [107].log_data[29].valid := 1, [107].log_data[30].min := 1.0, [107].log_data[30].max := 1.0, [107].log_data[30].total := 3600.0, [107].log_data[30].time := 3600.0, [107].log_data[30].valid := 1, [107].log_data[31].max := 1.0, [107].log_data[31].total := 1629.998, [107].log_data[31].time := 3600.0, [107].log_data[31].maxminute := 6, [107].log_data[31].valid := 1, [107].log_data[32].max := 1.0, [107].log_data[32].total := 1440.498, [107].log_data[32].time := 3600.0, [107].log_data[32].minminute := 5, [107].log_data[32].valid := 1, [107].log_data[33].time := 3600.0, [107].log_data[33].valid := 1, [107].log_data[34].time := 3600.0, [107].log_data[34].valid := 1, [107].log_data[35].max := 1.0, [107].log_data[35].total := 1629.7471, [107].log_data[35].time := 3600.0, [107].log_data[35].maxminute := 1, [107].log_data[35].valid := 1, [107].log_data[36].max := 1.0, [107].log_data[36].total := 1440.7471, [107].log_data[36].time := 3600.0, [107].log_data[36].valid := 1, [107].log_data[37].max := 7.2258115, [107].log_data[37].total := 3544.7075, [107].log_data[37].time := 3600.0, [107].log_data[37].maxminute := 15, [107].log_data[37].valid := 1, [107].log_data[38].time := 3600.0, [107].log_data[38].valid := 1, [107].log_data[39].min := 0.99541295, [107].log_data[39].max := 1.0212055, [107].log_data[39].total := 3608.5706, [107].log_data[39].time := 3600.0, [107].log_data[39].minminute := 4, [107].log_data[39].maxminute := 17, [107].log_data[39].valid := 1, [107].log_data[40].min := 7.58905, [107].log_data[40].max := 7.609111, [107].log_data[40].total := 27367.479, [107].log_data[40].time := 3600.0, [107].log_data[40].minminute := 20, [107].log_data[40].maxminute := 24, [107].log_data[40].valid := 1, [107].log_data[41].min := 0.02273633, [107].log_data[41].max := 0.023325196, [107].log_data[41].total := 82.74008, [107].log_data[41].time := 3600.0, [107].log_data[41].minminute := 1, [107].log_data[41].maxminute := 16,
        [107].log_data[41].valid := 1, [107].log_data[42].min := 2.2918782, [107].log_data[42].max := 2.296236, [107].log_data[42].total := 8259.035, [107].log_data[42].time := 3600.0, [107].log_data[42].minminute := 18, [107].log_data[42].maxminute := 39, [107].log_data[42].valid := 1, [107].log_data[43].min := -0.27999878, [107].log_data[43].max := -0.26000214, [107].log_data[43].total := -946.35706, [107].log_data[43].time := 3600.0, [107].log_data[43].valid := 1, [107].log_data[44].min := -0.3199997, [107].log_data[44].max := -0.30000305, [107].log_data[44].total := -1080.1161, [107].log_data[44].time := 3600.0, [107].log_data[44].valid := 1, [107].log_data[45].time := 3600.0, [107].log_data[45].valid := 1, [107].log_data[46].time := 3600.0, [107].log_data[46].valid := 1, [107].log_data[47].time := 3600.0, [107].log_data[47].valid := 1, [107].log_data[48].min := 6.578031, [107].log_data[48].max := 6.9009304, [107].log_data[48].total := 24185.686, [107].log_data[48].time := 3600.0, [107].log_data[48].minminute := 44, [107].log_data[48].maxminute := 20, [107].log_data[48].valid := 1, [107].log_data[49].min := 6.67564, [107].log_data[49].max := 9.43, [107].log_data[49].total := 28988.332, [107].log_data[49].time := 3600.0, [107].log_data[49].minminute := 45, [107].log_data[49].maxminute := 9, [107].log_data[49].valid := 1, [107].log_data[50].min := 1.9089923, [107].log_data[50].max := 2.0148718, [107].log_data[50].total := 7088.5483, [107].log_data[50].time := 3600.0, [107].log_data[50].minminute := 16, [107].log_data[50].maxminute := 25, [107].log_data[50].valid := 1, [107].log_data[51].time := 3600.0, [107].log_data[51].valid := 1, [107].log_data[52].min := -2.880005, [107].log_data[52].max := 0.11999512, [107].log_data[52].total := -7690.2197, [107].log_data[52].time := 3600.0, [107].log_data[52].minminute := 6, [107].log_data[52].maxminute := 5, [107].log_data[52].valid := 1, [107].log_data[53].min := -2.5200043, [107].log_data[53].max := 0.22000122, [107].log_data[53].total := -7233.3394, [107].log_data[53].time := 3600.0, [107].log_data[53].minminute := 4, [107].log_data[53].maxminute := 1,
        [107].log_data[53].valid := 1, [107].log_data[54].max := 0.5535, [107].log_data[54].total := 1217.4894, [107].log_data[54].time := 3600.0, [107].log_data[54].minminute := 5, [107].log_data[54].maxminute := 27, [107].log_data[54].valid := 1, [107].log_data[55].max := 0.525, [107].log_data[55].total := 1216.9321, [107].log_data[55].time := 3600.0, [107].log_data[55].maxminute := 1, [107].log_data[55].valid := 1, [107].log_data[56].min := 0.15953897, [107].log_data[56].max := 0.15993154, [107].log_data[56].total := 574.8502, [107].log_data[56].time := 3600.0, [107].log_data[56].minminute := 18, [107].log_data[56].maxminute := 3, [107].log_data[56].valid := 1, [107].log_data[57].min := 0.22710244, [107].log_data[57].max := 0.22926167, [107].log_data[57].total := 823.078, [107].log_data[57].time := 3600.0, [107].log_data[57].minminute := 56, [107].log_data[57].maxminute := 40, [107].log_data[57].valid := 1, [107].log_data[58].time := 3600.0, [107].log_data[58].valid := 1, [107].log_data[59].time := 3600.0, [107].log_data[59].valid := 1, [107].log_data[60].valid := 1, [107].log_data[61].valid := 1, [107].log_data[62].valid := 1, [107].log_data[63].valid := 1, [107].log_data[64].valid := 1, [107].log_data[65].valid := 1, [107].log_data[66].valid := 1, [107].log_data[67].valid := 1, [107].log_data[68].valid := 1, [107].log_data[69].valid := 1, [107].log_data[70].valid := 1, [107].log_data[71].valid := 1, [107].log_data[72].valid := 1, [107].log_data[73].valid := 1, [107].log_data[74].valid := 1, [107].log_data[75].valid := 1, [107].log_data[76].valid := 1, [107].log_data[77].valid := 1, [107].log_data[78].valid := 1, [107].log_data[79].valid := 1, [107].log_data[80].valid := 1, [107].log_data[81].valid := 1, [107].log_data[82].valid := 1, [107].log_data[83].valid := 1, [107].log_data[84].valid := 1, [107].log_data[85].valid := 1, [107].log_data[86].valid := 1, [107].log_data[87].valid := 1, [107].log_data[88].valid := 1, [107].log_data[89].valid := 1,
        [107].log_data[90].valid := 1, [107].log_data[91].valid := 1, [107].log_data[92].valid := 1, [107].log_data[93].valid := 1, [107].log_data[94].valid := 1, [107].log_data[95].valid := 1, [107].log_data[96].valid := 1, [107].log_data[97].valid := 1, [107].log_data[98].valid := 1, [107].log_data[99].valid := 1, [107].log_data[100].valid := 1, [107].log_data[101].valid := 1, [107].log_data[102].valid := 1, [107].log_data[103].valid := 1, [107].log_data[104].valid := 1, [107].log_data[105].valid := 1, [107].log_data[106].valid := 1, [107].log_data[107].valid := 1, [107].log_data[108].valid := 1, [107].log_data[109].valid := 1, [107].log_data[110].valid := 1, [107].log_data[111].valid := 1, [107].log_data[112].valid := 1, [107].log_data[113].valid := 1, [107].log_data[114].valid := 1, [107].log_data[115].valid := 1, [107].log_data[116].valid := 1, [107].log_data[117].valid := 1, [107].log_data[118].valid := 1, [107].log_data[119].valid := 1, [107].log_data[120].valid := 1, [107].log_data[121].valid := 1, [107].log_data[122].valid := 1, [107].log_data[123].valid := 1, [107].log_data[124].valid := 1, [107].time.Year := 2023, [107].time.Month := 1, [107].time.Day := 17, [107].time.Hour := 14, [107].time.Minute := 59, [107].time.Second := 59, [108].log_data[0].min := 1.0, [108].log_data[0].max := 1.0, [108].log_data[0].total := 3600.0, [108].log_data[0].time := 3600.0, [108].log_data[0].valid := 1, [108].log_data[1].time := 3600.0, [108].log_data[1].valid := 1, [108].log_data[2].time := 3600.0, [108].log_data[2].valid := 1, [108].log_data[3].time := 3600.0, [108].log_data[3].valid := 1, [108].log_data[4].time := 3600.0, [108].log_data[4].valid := 1, [108].log_data[5].time := 3600.0, [108].log_data[5].valid := 1, [108].log_data[6].time := 3600.0, [108].log_data[6].valid := 1, [108].log_data[7].time := 3600.0, [108].log_data[7].valid := 1,
        [108].log_data[8].min := 1.0, [108].log_data[8].max := 1.0, [108].log_data[8].total := 3600.0, [108].log_data[8].time := 3600.0, [108].log_data[8].valid := 1, [108].log_data[9].min := 1.0, [108].log_data[9].max := 1.0, [108].log_data[9].total := 3600.0, [108].log_data[9].time := 3600.0, [108].log_data[9].valid := 1, [108].log_data[10].min := 1.0, [108].log_data[10].max := 1.0, [108].log_data[10].total := 3600.0, [108].log_data[10].time := 3600.0, [108].log_data[10].valid := 1, [108].log_data[11].time := 3600.0, [108].log_data[11].valid := 1, [108].log_data[12].min := 1.0, [108].log_data[12].max := 1.0, [108].log_data[12].total := 3600.0, [108].log_data[12].time := 3600.0, [108].log_data[12].valid := 1, [108].log_data[13].min := 1.0, [108].log_data[13].max := 1.0, [108].log_data[13].total := 3600.0, [108].log_data[13].time := 3600.0, [108].log_data[13].valid := 1, [108].log_data[14].time := 3600.0, [108].log_data[14].valid := 1, [108].log_data[15].time := 3600.0, [108].log_data[15].valid := 1, [108].log_data[16].time := 3600.0, [108].log_data[16].valid := 1, [108].log_data[17].min := 1.0, [108].log_data[17].max := 1.0, [108].log_data[17].total := 3600.0, [108].log_data[17].time := 3600.0, [108].log_data[17].valid := 1, [108].log_data[18].time := 3600.0, [108].log_data[18].valid := 1, [108].log_data[19].time := 3600.0, [108].log_data[19].valid := 1, [108].log_data[20].time := 3600.0, [108].log_data[20].valid := 1, [108].log_data[21].min := 1.0, [108].log_data[21].max := 1.0, [108].log_data[21].total := 3600.0, [108].log_data[21].time := 3600.0, [108].log_data[21].valid := 1, [108].log_data[22].time := 3600.0, [108].log_data[22].valid := 1, [108].log_data[23].time := 3600.0, [108].log_data[23].valid := 1, [108].log_data[24].time := 3600.0, [108].log_data[24].valid := 1, [108].log_data[25].time := 3600.0, [108].log_data[25].valid := 1, [108].log_data[26].time := 3600.0, [108].log_data[26].valid := 1, [108].log_data[27].time := 3600.0,
        [108].log_data[27].valid := 1, [108].log_data[28].time := 3600.0, [108].log_data[28].valid := 1, [108].log_data[29].min := 1.0, [108].log_data[29].max := 1.0, [108].log_data[29].total := 3600.0, [108].log_data[29].time := 3600.0, [108].log_data[29].valid := 1, [108].log_data[30].min := 1.0, [108].log_data[30].max := 1.0, [108].log_data[30].total := 3600.0, [108].log_data[30].time := 3600.0, [108].log_data[30].valid := 1, [108].log_data[31].max := 1.0, [108].log_data[31].total := 1564.2471, [108].log_data[31].time := 3600.0, [108].log_data[31].maxminute := 9, [108].log_data[31].valid := 1, [108].log_data[32].max := 1.0, [108].log_data[32].total := 1594.749, [108].log_data[32].time := 3600.0, [108].log_data[32].minminute := 8, [108].log_data[32].valid := 1, [108].log_data[33].time := 3600.0, [108].log_data[33].valid := 1, [108].log_data[34].time := 3600.0, [108].log_data[34].valid := 1, [108].log_data[35].max := 1.0, [108].log_data[35].total := 1629.998, [108].log_data[35].time := 3600.0, [108].log_data[35].maxminute := 5, [108].log_data[35].valid := 1, [108].log_data[36].max := 1.0, [108].log_data[36].total := 1440.2471, [108].log_data[36].time := 3600.0, [108].log_data[36].minminute := 3, [108].log_data[36].valid := 1, [108].log_data[37].time := 3600.0, [108].log_data[37].valid := 1, [108].log_data[38].time := 3600.0, [108].log_data[38].valid := 1, [108].log_data[39].min := 0.9956484, [108].log_data[39].max := 1.0055416, [108].log_data[39].total := 3604.5186, [108].log_data[39].time := 3600.0, [108].log_data[39].minminute := 52, [108].log_data[39].maxminute := 15, [108].log_data[39].valid := 1, [108].log_data[40].min := 7.5775075, [108].log_data[40].max := 7.6093855, [108].log_data[40].total := 27366.121, [108].log_data[40].time := 3600.0, [108].log_data[40].minminute := 56, [108].log_data[40].maxminute := 22, [108].log_data[40].valid := 1, [108].log_data[41].min := 0.02273633, [108].log_data[41].max := 0.023128908, [108].log_data[41].total := 82.66988, [108].log_data[41].time := 3600.0, [108].log_data[41].valid := 1,
        [108].log_data[42].min := 2.291407, [108].log_data[42].max := 2.296236, [108].log_data[42].total := 8259.108, [108].log_data[42].time := 3600.0, [108].log_data[42].minminute := 18, [108].log_data[42].maxminute := 33, [108].log_data[42].valid := 1, [108].log_data[43].min := -0.27999878, [108].log_data[43].max := -0.26000214, [108].log_data[43].total := -937.62756, [108].log_data[43].time := 3600.0, [108].log_data[43].valid := 1, [108].log_data[44].min := -0.30000305, [108].log_data[44].max := -0.27999878, [108].log_data[44].total := -1080.0709, [108].log_data[44].time := 3600.0, [108].log_data[44].maxminute := 14, [108].log_data[44].valid := 1, [108].log_data[45].time := 3600.0, [108].log_data[45].valid := 1, [108].log_data[46].time := 3600.0, [108].log_data[46].valid := 1, [108].log_data[47].time := 3600.0, [108].log_data[47].valid := 1, [108].log_data[48].min := 6.740717, [108].log_data[48].max := 6.7998004, [108].log_data[48].total := 24325.684, [108].log_data[48].time := 3600.0, [108].log_data[48].minminute := 59, [108].log_data[48].valid := 1, [108].log_data[49].min := 8.262461, [108].log_data[49].max := 9.402521, [108].log_data[49].total := 33049.754, [108].log_data[49].time := 3600.0, [108].log_data[49].maxminute := 51, [108].log_data[49].valid := 1, [108].log_data[50].min := 1.8724821, [108].log_data[50].max := 1.9736506, [108].log_data[50].total := 6935.5737, [108].log_data[50].time := 3600.0, [108].log_data[50].minminute := 59, [108].log_data[50].valid := 1, [108].log_data[51].time := 3600.0, [108].log_data[51].valid := 1, [108].log_data[52].min := -2.959999, [108].log_data[52].max := 0.11999512, [108].log_data[52].total := -7974.48, [108].log_data[52].time := 3600.0, [108].log_data[52].minminute := 31, [108].log_data[52].maxminute := 8, [108].log_data[52].valid := 1, [108].log_data[53].min := -2.5200043, [108].log_data[53].max := 0.19999695, [108].log_data[53].total := -7278.168, [108].log_data[53].time := 3600.0, [108].log_data[53].minminute := 6, [108].log_data[53].maxminute := 36, [108].log_data[53].valid := 1, [108].log_data[54].max := 0.5295, [108].log_data[54].total := 1254.3359,
        [108].log_data[54].time := 3600.0, [108].log_data[54].minminute := 8, [108].log_data[54].maxminute := 10, [108].log_data[54].valid := 1, [108].log_data[55].max := 0.5255, [108].log_data[55].total := 1216.9525, [108].log_data[55].time := 3600.0, [108].log_data[55].minminute := 3, [108].log_data[55].maxminute := 47, [108].log_data[55].valid := 1, [108].log_data[56].min := 0.1594997, [108].log_data[56].max := 0.15993154, [108].log_data[56].total := 574.8085, [108].log_data[56].time := 3600.0, [108].log_data[56].minminute := 41, [108].log_data[56].maxminute := 12, [108].log_data[56].valid := 1, [108].log_data[57].min := 0.2271417, [108].log_data[57].max := 0.22753428, [108].log_data[57].total := 818.2298, [108].log_data[57].time := 3600.0, [108].log_data[57].maxminute := 37, [108].log_data[57].valid := 1, [108].log_data[58].time := 3600.0, [108].log_data[58].valid := 1, [108].log_data[59].time := 3600.0, [108].log_data[59].valid := 1, [108].log_data[60].valid := 1, [108].log_data[61].valid := 1, [108].log_data[62].valid := 1, [108].log_data[63].valid := 1, [108].log_data[64].valid := 1, [108].log_data[65].valid := 1, [108].log_data[66].valid := 1, [108].log_data[67].valid := 1, [108].log_data[68].valid := 1, [108].log_data[69].valid := 1, [108].log_data[70].valid := 1, [108].log_data[71].valid := 1, [108].log_data[72].valid := 1, [108].log_data[73].valid := 1, [108].log_data[74].valid := 1, [108].log_data[75].valid := 1, [108].log_data[76].valid := 1, [108].log_data[77].valid := 1, [108].log_data[78].valid := 1, [108].log_data[79].valid := 1, [108].log_data[80].valid := 1, [108].log_data[81].valid := 1, [108].log_data[82].valid := 1, [108].log_data[83].valid := 1, [108].log_data[84].valid := 1, [108].log_data[85].valid := 1, [108].log_data[86].valid := 1, [108].log_data[87].valid := 1, [108].log_data[88].valid := 1, [108].log_data[89].valid := 1, [108].log_data[90].valid := 1, [108].log_data[91].valid := 1, [108].log_data[92].valid := 1,
        [108].log_data[93].valid := 1, [108].log_data[94].valid := 1, [108].log_data[95].valid := 1, [108].log_data[96].valid := 1, [108].log_data[97].valid := 1, [108].log_data[98].valid := 1, [108].log_data[99].valid := 1, [108].log_data[100].valid := 1, [108].log_data[101].valid := 1, [108].log_data[102].valid := 1, [108].log_data[103].valid := 1, [108].log_data[104].valid := 1, [108].log_data[105].valid := 1, [108].log_data[106].valid := 1, [108].log_data[107].valid := 1, [108].log_data[108].valid := 1, [108].log_data[109].valid := 1, [108].log_data[110].valid := 1, [108].log_data[111].valid := 1, [108].log_data[112].valid := 1, [108].log_data[113].valid := 1, [108].log_data[114].valid := 1, [108].log_data[115].valid := 1, [108].log_data[116].valid := 1, [108].log_data[117].valid := 1, [108].log_data[118].valid := 1, [108].log_data[119].valid := 1, [108].log_data[120].valid := 1, [108].log_data[121].valid := 1, [108].log_data[122].valid := 1, [108].log_data[123].valid := 1, [108].log_data[124].valid := 1, [108].time.Year := 2023, [108].time.Month := 1, [108].time.Day := 17, [108].time.Hour := 15, [108].time.Minute := 59, [108].time.Second := 59, [109].log_data[0].min := 1.0, [109].log_data[0].max := 1.0, [109].log_data[0].total := 3600.0, [109].log_data[0].time := 3600.0, [109].log_data[0].valid := 1, [109].log_data[1].max := 1.0, [109].log_data[1].total := 532.5, [109].log_data[1].time := 3600.0, [109].log_data[1].maxminute := 21, [109].log_data[1].valid := 1, [109].log_data[2].max := 1.0, [109].log_data[2].total := 529.0, [109].log_data[2].time := 3600.0, [109].log_data[2].maxminute := 21, [109].log_data[2].valid := 1, [109].log_data[3].time := 3600.0, [109].log_data[3].valid := 1, [109].log_data[4].time := 3600.0, [109].log_data[4].valid := 1, [109].log_data[5].max := 1.0, [109].log_data[5].total := 241.5, [109].log_data[5].time := 3600.0,
        [109].log_data[5].maxminute := 23, [109].log_data[5].valid := 1, [109].log_data[6].time := 3600.0, [109].log_data[6].valid := 1, [109].log_data[7].time := 3600.0, [109].log_data[7].valid := 1, [109].log_data[8].min := 1.0, [109].log_data[8].max := 1.0, [109].log_data[8].total := 3600.0, [109].log_data[8].time := 3600.0, [109].log_data[8].valid := 1, [109].log_data[9].min := 1.0, [109].log_data[9].max := 1.0, [109].log_data[9].total := 3600.0, [109].log_data[9].time := 3600.0, [109].log_data[9].valid := 1, [109].log_data[10].min := 1.0, [109].log_data[10].max := 1.0, [109].log_data[10].total := 3600.0, [109].log_data[10].time := 3600.0, [109].log_data[10].valid := 1, [109].log_data[11].time := 3600.0, [109].log_data[11].valid := 1, [109].log_data[12].min := 1.0, [109].log_data[12].max := 1.0, [109].log_data[12].total := 3600.0, [109].log_data[12].time := 3600.0, [109].log_data[12].valid := 1, [109].log_data[13].min := 1.0, [109].log_data[13].max := 1.0, [109].log_data[13].total := 3600.0, [109].log_data[13].time := 3600.0, [109].log_data[13].valid := 1, [109].log_data[14].time := 3600.0, [109].log_data[14].valid := 1, [109].log_data[15].time := 3600.0, [109].log_data[15].valid := 1, [109].log_data[16].time := 3600.0, [109].log_data[16].valid := 1, [109].log_data[17].min := 1.0, [109].log_data[17].max := 1.0, [109].log_data[17].total := 3600.0, [109].log_data[17].time := 3600.0, [109].log_data[17].valid := 1, [109].log_data[18].time := 3600.0, [109].log_data[18].valid := 1, [109].log_data[19].time := 3600.0, [109].log_data[19].valid := 1, [109].log_data[20].time := 3600.0, [109].log_data[20].valid := 1, [109].log_data[21].min := 1.0, [109].log_data[21].max := 1.0, [109].log_data[21].total := 3600.0, [109].log_data[21].time := 3600.0, [109].log_data[21].valid := 1, [109].log_data[22].time := 3600.0, [109].log_data[22].valid := 1, [109].log_data[23].time := 3600.0, [109].log_data[23].valid := 1, [109].log_data[24].time := 3600.0,
        [109].log_data[24].valid := 1, [109].log_data[25].time := 3600.0, [109].log_data[25].valid := 1, [109].log_data[26].time := 3600.0, [109].log_data[26].valid := 1, [109].log_data[27].time := 3600.0, [109].log_data[27].valid := 1, [109].log_data[28].time := 3600.0, [109].log_data[28].valid := 1, [109].log_data[29].min := 1.0, [109].log_data[29].max := 1.0, [109].log_data[29].total := 3600.0, [109].log_data[29].time := 3600.0, [109].log_data[29].valid := 1, [109].log_data[30].min := 1.0, [109].log_data[30].max := 1.0, [109].log_data[30].total := 3600.0, [109].log_data[30].time := 3600.0, [109].log_data[30].valid := 1, [109].log_data[31].max := 1.0, [109].log_data[31].total := 1440.7471, [109].log_data[31].time := 3600.0, [109].log_data[31].minminute := 1, [109].log_data[31].valid := 1, [109].log_data[32].max := 1.0, [109].log_data[32].total := 1629.7471, [109].log_data[32].time := 3600.0, [109].log_data[32].maxminute := 2, [109].log_data[32].valid := 1, [109].log_data[33].time := 3600.0, [109].log_data[33].valid := 1, [109].log_data[34].time := 3600.0, [109].log_data[34].valid := 1, [109].log_data[35].max := 1.0, [109].log_data[35].total := 1629.498, [109].log_data[35].time := 3600.0, [109].log_data[35].maxminute := 8, [109].log_data[35].valid := 1, [109].log_data[36].max := 1.0, [109].log_data[36].total := 1488.5, [109].log_data[36].time := 3600.0, [109].log_data[36].minminute := 6, [109].log_data[36].valid := 1, [109].log_data[37].max := 7.590914, [109].log_data[37].total := 3491.166, [109].log_data[37].time := 3600.0, [109].log_data[37].maxminute := 22, [109].log_data[37].valid := 1, [109].log_data[38].time := 3600.0, [109].log_data[38].valid := 1, [109].log_data[39].min := 0.9947063, [109].log_data[39].max := 1.0219122, [109].log_data[39].total := 3607.0737, [109].log_data[39].time := 3600.0, [109].log_data[39].minminute := 30, [109].log_data[39].maxminute := 24, [109].log_data[39].valid := 1, [109].log_data[40].min := 7.5802555, [109].log_data[40].max := 7.6121335, [109].log_data[40].total := 27369.365,
        [109].log_data[40].time := 3600.0, [109].log_data[40].minminute := 7, [109].log_data[40].maxminute := 9, [109].log_data[40].valid := 1, [109].log_data[41].min := 0.02273633, [109].log_data[41].max := 0.023325196, [109].log_data[41].total := 82.5984, [109].log_data[41].time := 3600.0, [109].log_data[41].maxminute := 25, [109].log_data[41].valid := 1, [109].log_data[42].min := 2.2917604, [109].log_data[42].max := 2.296236, [109].log_data[42].total := 8259.09, [109].log_data[42].time := 3600.0, [109].log_data[42].minminute := 6, [109].log_data[42].maxminute := 32, [109].log_data[42].valid := 1, [109].log_data[43].min := -0.27999878, [109].log_data[43].max := -0.26000214, [109].log_data[43].total := -936.4781, [109].log_data[43].time := 3600.0, [109].log_data[43].valid := 1, [109].log_data[44].min := -0.30000305, [109].log_data[44].max := -0.27999878, [109].log_data[44].total := -1080.0409, [109].log_data[44].time := 3600.0, [109].log_data[44].valid := 1, [109].log_data[45].time := 3600.0, [109].log_data[45].valid := 1, [109].log_data[46].time := 3600.0, [109].log_data[46].valid := 1, [109].log_data[47].time := 3600.0, [109].log_data[47].valid := 1, [109].log_data[48].min := 6.5722604, [109].log_data[48].max := 6.9179688, [109].log_data[48].total := 24158.03, [109].log_data[48].time := 3600.0, [109].log_data[48].minminute := 50, [109].log_data[48].maxminute := 30, [109].log_data[48].valid := 1, [109].log_data[49].min := 6.6032085, [109].log_data[49].max := 9.401342, [109].log_data[49].total := 29461.006, [109].log_data[49].time := 3600.0, [109].log_data[49].minminute := 52, [109].log_data[49].valid := 1, [109].log_data[50].min := 1.8425672, [109].log_data[50].max := 1.9552777, [109].log_data[50].total := 6850.263, [109].log_data[50].time := 3600.0, [109].log_data[50].minminute := 22, [109].log_data[50].maxminute := 30, [109].log_data[50].valid := 1, [109].log_data[51].time := 3600.0, [109].log_data[51].valid := 1, [109].log_data[52].min := -2.959999, [109].log_data[52].max := 0.11999512, [109].log_data[52].total := -7772.408, [109].log_data[52].time := 3600.0, [109].log_data[52].minminute := 55,
        [109].log_data[52].maxminute := 1, [109].log_data[52].valid := 1, [109].log_data[53].min := -2.5200043, [109].log_data[53].max := 0.22000122, [109].log_data[53].total := -7459.609, [109].log_data[53].time := 3600.0, [109].log_data[53].minminute := 8, [109].log_data[53].maxminute := 39, [109].log_data[53].valid := 1, [109].log_data[54].max := 0.52349997, [109].log_data[54].total := 1217.3887, [109].log_data[54].time := 3600.0, [109].log_data[54].minminute := 1, [109].log_data[54].maxminute := 34, [109].log_data[54].valid := 1, [109].log_data[55].max := 0.5385, [109].log_data[55].total := 1238.6794, [109].log_data[55].time := 3600.0, [109].log_data[55].minminute := 6, [109].log_data[55].maxminute := 8, [109].log_data[55].valid := 1, [109].log_data[56].min := 0.15942119, [109].log_data[56].max := 0.15989229, [109].log_data[56].total := 574.62164, [109].log_data[56].time := 3600.0, [109].log_data[56].minminute := 38, [109].log_data[56].maxminute := 37, [109].log_data[56].valid := 1, [109].log_data[57].min := 0.22498251, [109].log_data[57].max := 0.22757353, [109].log_data[57].total := 817.41437, [109].log_data[57].time := 3600.0, [109].log_data[57].minminute := 59, [109].log_data[57].maxminute := 22, [109].log_data[57].valid := 1, [109].log_data[58].time := 3600.0, [109].log_data[58].valid := 1, [109].log_data[59].time := 3600.0, [109].log_data[59].valid := 1, [109].log_data[60].valid := 1, [109].log_data[61].valid := 1, [109].log_data[62].valid := 1, [109].log_data[63].valid := 1, [109].log_data[64].valid := 1, [109].log_data[65].valid := 1, [109].log_data[66].valid := 1, [109].log_data[67].valid := 1, [109].log_data[68].valid := 1, [109].log_data[69].valid := 1, [109].log_data[70].valid := 1, [109].log_data[71].valid := 1, [109].log_data[72].valid := 1, [109].log_data[73].valid := 1, [109].log_data[74].valid := 1, [109].log_data[75].valid := 1, [109].log_data[76].valid := 1, [109].log_data[77].valid := 1, [109].log_data[78].valid := 1, [109].log_data[79].valid := 1, [109].log_data[80].valid := 1,
        [109].log_data[81].valid := 1, [109].log_data[82].valid := 1, [109].log_data[83].valid := 1, [109].log_data[84].valid := 1, [109].log_data[85].valid := 1, [109].log_data[86].valid := 1, [109].log_data[87].valid := 1, [109].log_data[88].valid := 1, [109].log_data[89].valid := 1, [109].log_data[90].valid := 1, [109].log_data[91].valid := 1, [109].log_data[92].valid := 1, [109].log_data[93].valid := 1, [109].log_data[94].valid := 1, [109].log_data[95].valid := 1, [109].log_data[96].valid := 1, [109].log_data[97].valid := 1, [109].log_data[98].valid := 1, [109].log_data[99].valid := 1, [109].log_data[100].valid := 1, [109].log_data[101].valid := 1, [109].log_data[102].valid := 1, [109].log_data[103].valid := 1, [109].log_data[104].valid := 1, [109].log_data[105].valid := 1, [109].log_data[106].valid := 1, [109].log_data[107].valid := 1, [109].log_data[108].valid := 1, [109].log_data[109].valid := 1, [109].log_data[110].valid := 1, [109].log_data[111].valid := 1, [109].log_data[112].valid := 1, [109].log_data[113].valid := 1, [109].log_data[114].valid := 1, [109].log_data[115].valid := 1, [109].log_data[116].valid := 1, [109].log_data[117].valid := 1, [109].log_data[118].valid := 1, [109].log_data[119].valid := 1, [109].log_data[120].valid := 1, [109].log_data[121].valid := 1, [109].log_data[122].valid := 1, [109].log_data[123].valid := 1, [109].log_data[124].valid := 1, [109].time.Year := 2023, [109].time.Month := 1, [109].time.Day := 17, [109].time.Hour := 16, [109].time.Minute := 59, [109].time.Second := 59, [110].log_data[0].min := 1.0, [110].log_data[0].max := 1.0, [110].log_data[0].total := 3600.0, [110].log_data[0].time := 3600.0, [110].log_data[0].valid := 1, [110].log_data[1].time := 3600.0, [110].log_data[1].valid := 1, [110].log_data[2].time := 3600.0, [110].log_data[2].valid := 1, [110].log_data[3].time := 3600.0,
        [110].log_data[3].valid := 1, [110].log_data[4].time := 3600.0, [110].log_data[4].valid := 1, [110].log_data[5].time := 3600.0, [110].log_data[5].valid := 1, [110].log_data[6].time := 3600.0, [110].log_data[6].valid := 1, [110].log_data[7].time := 3600.0, [110].log_data[7].valid := 1, [110].log_data[8].min := 1.0, [110].log_data[8].max := 1.0, [110].log_data[8].total := 3600.0, [110].log_data[8].time := 3600.0, [110].log_data[8].valid := 1, [110].log_data[9].min := 1.0, [110].log_data[9].max := 1.0, [110].log_data[9].total := 3600.0, [110].log_data[9].time := 3600.0, [110].log_data[9].valid := 1, [110].log_data[10].min := 1.0, [110].log_data[10].max := 1.0, [110].log_data[10].total := 3600.0, [110].log_data[10].time := 3600.0, [110].log_data[10].valid := 1, [110].log_data[11].time := 3600.0, [110].log_data[11].valid := 1, [110].log_data[12].min := 1.0, [110].log_data[12].max := 1.0, [110].log_data[12].total := 3600.0, [110].log_data[12].time := 3600.0, [110].log_data[12].valid := 1, [110].log_data[13].min := 1.0, [110].log_data[13].max := 1.0, [110].log_data[13].total := 3600.0, [110].log_data[13].time := 3600.0, [110].log_data[13].valid := 1, [110].log_data[14].time := 3600.0, [110].log_data[14].valid := 1, [110].log_data[15].time := 3600.0, [110].log_data[15].valid := 1, [110].log_data[16].time := 3600.0, [110].log_data[16].valid := 1, [110].log_data[17].min := 1.0, [110].log_data[17].max := 1.0, [110].log_data[17].total := 3600.0, [110].log_data[17].time := 3600.0, [110].log_data[17].valid := 1, [110].log_data[18].time := 3600.0, [110].log_data[18].valid := 1, [110].log_data[19].time := 3600.0, [110].log_data[19].valid := 1, [110].log_data[20].time := 3600.0, [110].log_data[20].valid := 1, [110].log_data[21].min := 1.0, [110].log_data[21].max := 1.0, [110].log_data[21].total := 3600.0, [110].log_data[21].time := 3600.0, [110].log_data[21].valid := 1, [110].log_data[22].time := 3600.0, [110].log_data[22].valid := 1,
        [110].log_data[23].time := 3600.0, [110].log_data[23].valid := 1, [110].log_data[24].time := 3600.0, [110].log_data[24].valid := 1, [110].log_data[25].time := 3600.0, [110].log_data[25].valid := 1, [110].log_data[26].time := 3600.0, [110].log_data[26].valid := 1, [110].log_data[27].time := 3600.0, [110].log_data[27].valid := 1, [110].log_data[28].time := 3600.0, [110].log_data[28].valid := 1, [110].log_data[29].min := 1.0, [110].log_data[29].max := 1.0, [110].log_data[29].total := 3600.0, [110].log_data[29].time := 3600.0, [110].log_data[29].valid := 1, [110].log_data[30].min := 1.0, [110].log_data[30].max := 1.0, [110].log_data[30].total := 3600.0, [110].log_data[30].time := 3600.0, [110].log_data[30].valid := 1, [110].log_data[31].max := 1.0, [110].log_data[31].total := 1440.7471, [110].log_data[31].time := 3600.0, [110].log_data[31].minminute := 4, [110].log_data[31].valid := 1, [110].log_data[32].max := 1.0, [110].log_data[32].total := 1630.249, [110].log_data[32].time := 3600.0, [110].log_data[32].maxminute := 5, [110].log_data[32].valid := 1, [110].log_data[33].time := 3600.0, [110].log_data[33].valid := 1, [110].log_data[34].time := 3600.0, [110].log_data[34].valid := 1, [110].log_data[35].max := 1.0, [110].log_data[35].total := 1481.498, [110].log_data[35].time := 3600.0, [110].log_data[35].maxminute := 11, [110].log_data[35].valid := 1, [110].log_data[36].max := 1.0, [110].log_data[36].total := 1629.7471, [110].log_data[36].time := 3600.0, [110].log_data[36].valid := 1, [110].log_data[37].time := 3600.0, [110].log_data[37].valid := 1, [110].log_data[38].time := 3600.0, [110].log_data[38].valid := 1, [110].log_data[39].min := 0.9951773, [110].log_data[39].max := 1.0042459, [110].log_data[39].total := 3600.125, [110].log_data[39].time := 3600.0, [110].log_data[39].minminute := 8, [110].log_data[39].maxminute := 11, [110].log_data[39].valid := 1, [110].log_data[40].min := 7.579981, [110].log_data[40].max := 7.6162558, [110].log_data[40].total := 27366.463, [110].log_data[40].time := 3600.0,
        [110].log_data[40].minminute := 35, [110].log_data[40].maxminute := 39, [110].log_data[40].valid := 1, [110].log_data[41].min := 0.02273633, [110].log_data[41].max := 0.023128908, [110].log_data[41].total := 82.53889, [110].log_data[41].time := 3600.0, [110].log_data[41].valid := 1, [110].log_data[42].min := 2.2918782, [110].log_data[42].max := 2.2963536, [110].log_data[42].total := 8259.069, [110].log_data[42].time := 3600.0, [110].log_data[42].minminute := 10, [110].log_data[42].maxminute := 2, [110].log_data[42].valid := 1, [110].log_data[43].min := -0.27999878, [110].log_data[43].max := -0.26000214, [110].log_data[43].total := -936.4171, [110].log_data[43].time := 3600.0, [110].log_data[43].valid := 1, [110].log_data[44].min := -0.30000305, [110].log_data[44].max := -0.27999878, [110].log_data[44].total := -1080.081, [110].log_data[44].time := 3600.0, [110].log_data[44].maxminute := 2, [110].log_data[44].valid := 1, [110].log_data[45].time := 3600.0, [110].log_data[45].valid := 1, [110].log_data[46].time := 3600.0, [110].log_data[46].valid := 1, [110].log_data[47].time := 3600.0, [110].log_data[47].valid := 1, [110].log_data[48].min := 6.7179084, [110].log_data[48].max := 6.7984266, [110].log_data[48].total := 24322.104, [110].log_data[48].time := 3600.0, [110].log_data[48].maxminute := 6, [110].log_data[48].valid := 1, [110].log_data[49].min := 7.4364657, [110].log_data[49].max := 9.376806, [110].log_data[49].total := 32391.775, [110].log_data[49].time := 3600.0, [110].log_data[49].maxminute := 48, [110].log_data[49].valid := 1, [110].log_data[50].min := 1.8362074, [110].log_data[50].max := 1.9213586, [110].log_data[50].total := 6761.256, [110].log_data[50].time := 3600.0, [110].log_data[50].minminute := 59, [110].log_data[50].valid := 1, [110].log_data[51].time := 3600.0, [110].log_data[51].valid := 1, [110].log_data[52].min := -2.9199982, [110].log_data[52].max := 0.11999512, [110].log_data[52].total := -7740.9526, [110].log_data[52].time := 3600.0, [110].log_data[52].minminute := 58, [110].log_data[52].maxminute := 4, [110].log_data[52].valid := 1, [110].log_data[53].min := -2.5600052,
        [110].log_data[53].max := 0.16000366, [110].log_data[53].total := -7439.1753, [110].log_data[53].time := 3600.0, [110].log_data[53].minminute := 35, [110].log_data[53].valid := 1, [110].log_data[54].max := 0.532, [110].log_data[54].total := 1217.3245, [110].log_data[54].time := 3600.0, [110].log_data[54].minminute := 4, [110].log_data[54].maxminute := 58, [110].log_data[54].valid := 1, [110].log_data[55].max := 0.52900004, [110].log_data[55].total := 1233.0444, [110].log_data[55].time := 3600.0, [110].log_data[55].maxminute := 43, [110].log_data[55].valid := 1, [110].log_data[56].min := 0.15934268, [110].log_data[56].max := 0.15989229, [110].log_data[56].total := 574.5449, [110].log_data[56].time := 3600.0, [110].log_data[56].minminute := 39, [110].log_data[56].maxminute := 10, [110].log_data[56].valid := 1, [110].log_data[57].min := 0.224904, [110].log_data[57].max := 0.22533584, [110].log_data[57].total := 810.2705, [110].log_data[57].time := 3600.0, [110].log_data[57].minminute := 3, [110].log_data[57].maxminute := 33, [110].log_data[57].valid := 1, [110].log_data[58].time := 3600.0, [110].log_data[58].valid := 1, [110].log_data[59].time := 3600.0, [110].log_data[59].valid := 1, [110].log_data[60].valid := 1, [110].log_data[61].valid := 1, [110].log_data[62].valid := 1, [110].log_data[63].valid := 1, [110].log_data[64].valid := 1, [110].log_data[65].valid := 1, [110].log_data[66].valid := 1, [110].log_data[67].valid := 1, [110].log_data[68].valid := 1, [110].log_data[69].valid := 1, [110].log_data[70].valid := 1, [110].log_data[71].valid := 1, [110].log_data[72].valid := 1, [110].log_data[73].valid := 1, [110].log_data[74].valid := 1, [110].log_data[75].valid := 1, [110].log_data[76].valid := 1, [110].log_data[77].valid := 1, [110].log_data[78].valid := 1, [110].log_data[79].valid := 1, [110].log_data[80].valid := 1, [110].log_data[81].valid := 1, [110].log_data[82].valid := 1, [110].log_data[83].valid := 1, [110].log_data[84].valid := 1, [110].log_data[85].valid := 1,
        [110].log_data[86].valid := 1, [110].log_data[87].valid := 1, [110].log_data[88].valid := 1, [110].log_data[89].valid := 1, [110].log_data[90].valid := 1, [110].log_data[91].valid := 1, [110].log_data[92].valid := 1, [110].log_data[93].valid := 1, [110].log_data[94].valid := 1, [110].log_data[95].valid := 1, [110].log_data[96].valid := 1, [110].log_data[97].valid := 1, [110].log_data[98].valid := 1, [110].log_data[99].valid := 1, [110].log_data[100].valid := 1, [110].log_data[101].valid := 1, [110].log_data[102].valid := 1, [110].log_data[103].valid := 1, [110].log_data[104].valid := 1, [110].log_data[105].valid := 1, [110].log_data[106].valid := 1, [110].log_data[107].valid := 1, [110].log_data[108].valid := 1, [110].log_data[109].valid := 1, [110].log_data[110].valid := 1, [110].log_data[111].valid := 1, [110].log_data[112].valid := 1, [110].log_data[113].valid := 1, [110].log_data[114].valid := 1, [110].log_data[115].valid := 1, [110].log_data[116].valid := 1, [110].log_data[117].valid := 1, [110].log_data[118].valid := 1, [110].log_data[119].valid := 1, [110].log_data[120].valid := 1, [110].log_data[121].valid := 1, [110].log_data[122].valid := 1, [110].log_data[123].valid := 1, [110].log_data[124].valid := 1, [110].time.Year := 2023, [110].time.Month := 1, [110].time.Day := 17, [110].time.Hour := 17, [110].time.Minute := 59, [110].time.Second := 59, [111].log_data[0].min := 1.0, [111].log_data[0].max := 1.0, [111].log_data[0].total := 3600.0, [111].log_data[0].time := 3600.0, [111].log_data[0].valid := 1, [111].log_data[1].max := 1.0, [111].log_data[1].total := 572.0, [111].log_data[1].time := 3600.0, [111].log_data[1].maxminute := 13, [111].log_data[1].valid := 1, [111].log_data[2].max := 1.0, [111].log_data[2].total := 568.5, [111].log_data[2].time := 3600.0, [111].log_data[2].maxminute := 13, [111].log_data[2].valid := 1,
        [111].log_data[3].time := 3600.0, [111].log_data[3].valid := 1, [111].log_data[4].time := 3600.0, [111].log_data[4].valid := 1, [111].log_data[5].max := 1.0, [111].log_data[5].total := 243.5, [111].log_data[5].time := 3600.0, [111].log_data[5].maxminute := 15, [111].log_data[5].valid := 1, [111].log_data[6].time := 3600.0, [111].log_data[6].valid := 1, [111].log_data[7].time := 3600.0, [111].log_data[7].valid := 1, [111].log_data[8].min := 1.0, [111].log_data[8].max := 1.0, [111].log_data[8].total := 3600.0, [111].log_data[8].time := 3600.0, [111].log_data[8].valid := 1, [111].log_data[9].min := 1.0, [111].log_data[9].max := 1.0, [111].log_data[9].total := 3600.0, [111].log_data[9].time := 3600.0, [111].log_data[9].valid := 1, [111].log_data[10].min := 1.0, [111].log_data[10].max := 1.0, [111].log_data[10].total := 3600.0, [111].log_data[10].time := 3600.0, [111].log_data[10].valid := 1, [111].log_data[11].time := 3600.0, [111].log_data[11].valid := 1, [111].log_data[12].min := 1.0, [111].log_data[12].max := 1.0, [111].log_data[12].total := 3600.0, [111].log_data[12].time := 3600.0, [111].log_data[12].valid := 1, [111].log_data[13].min := 1.0, [111].log_data[13].max := 1.0, [111].log_data[13].total := 3600.0, [111].log_data[13].time := 3600.0, [111].log_data[13].valid := 1, [111].log_data[14].time := 3600.0, [111].log_data[14].valid := 1, [111].log_data[15].time := 3600.0, [111].log_data[15].valid := 1, [111].log_data[16].time := 3600.0, [111].log_data[16].valid := 1, [111].log_data[17].min := 1.0, [111].log_data[17].max := 1.0, [111].log_data[17].total := 3600.0, [111].log_data[17].time := 3600.0, [111].log_data[17].valid := 1, [111].log_data[18].time := 3600.0, [111].log_data[18].valid := 1, [111].log_data[19].time := 3600.0, [111].log_data[19].valid := 1, [111].log_data[20].time := 3600.0, [111].log_data[20].valid := 1, [111].log_data[21].min := 1.0, [111].log_data[21].max := 1.0, [111].log_data[21].total := 3600.0,
        [111].log_data[21].time := 3600.0, [111].log_data[21].valid := 1, [111].log_data[22].time := 3600.0, [111].log_data[22].valid := 1, [111].log_data[23].time := 3600.0, [111].log_data[23].valid := 1, [111].log_data[24].time := 3600.0, [111].log_data[24].valid := 1, [111].log_data[25].time := 3600.0, [111].log_data[25].valid := 1, [111].log_data[26].time := 3600.0, [111].log_data[26].valid := 1, [111].log_data[27].time := 3600.0, [111].log_data[27].valid := 1, [111].log_data[28].time := 3600.0, [111].log_data[28].valid := 1, [111].log_data[29].min := 1.0, [111].log_data[29].max := 1.0, [111].log_data[29].total := 3600.0, [111].log_data[29].time := 3600.0, [111].log_data[29].valid := 1, [111].log_data[30].min := 1.0, [111].log_data[30].max := 1.0, [111].log_data[30].total := 3600.0, [111].log_data[30].time := 3600.0, [111].log_data[30].valid := 1, [111].log_data[31].max := 1.0, [111].log_data[31].total := 1530.249, [111].log_data[31].time := 3600.0, [111].log_data[31].minminute := 7, [111].log_data[31].valid := 1, [111].log_data[32].max := 1.0, [111].log_data[32].total := 1628.998, [111].log_data[32].time := 3600.0, [111].log_data[32].maxminute := 8, [111].log_data[32].valid := 1, [111].log_data[33].time := 3600.0, [111].log_data[33].valid := 1, [111].log_data[34].time := 3600.0, [111].log_data[34].valid := 1, [111].log_data[35].max := 1.0, [111].log_data[35].total := 1440.7471, [111].log_data[35].time := 3600.0, [111].log_data[35].minminute := 2, [111].log_data[35].valid := 1, [111].log_data[36].max := 1.0, [111].log_data[36].total := 1629.7471, [111].log_data[36].time := 3600.0, [111].log_data[36].maxminute := 3, [111].log_data[36].valid := 1, [111].log_data[37].max := 7.3773484, [111].log_data[37].total := 3648.963, [111].log_data[37].time := 3600.0, [111].log_data[37].maxminute := 14, [111].log_data[37].valid := 1, [111].log_data[38].time := 3600.0, [111].log_data[38].valid := 1, [111].log_data[39].min := 0.9951773, [111].log_data[39].max := 1.0212055, [111].log_data[39].total := 3607.0789,
        [111].log_data[39].time := 3600.0, [111].log_data[39].minminute := 2, [111].log_data[39].maxminute := 20, [111].log_data[39].valid := 1, [111].log_data[40].min := 7.590149, [111].log_data[40].max := 7.6107597, [111].log_data[40].total := 27368.23, [111].log_data[40].time := 3600.0, [111].log_data[40].minminute := 9, [111].log_data[40].maxminute := 11, [111].log_data[40].valid := 1, [111].log_data[41].min := 0.02273633, [111].log_data[41].max := 0.023325196, [111].log_data[41].total := 82.52646, [111].log_data[41].time := 3600.0, [111].log_data[41].maxminute := 18, [111].log_data[41].valid := 1, [111].log_data[42].min := 2.2917604, [111].log_data[42].max := 2.296118, [111].log_data[42].total := 8258.996, [111].log_data[42].time := 3600.0, [111].log_data[42].minminute := 1, [111].log_data[42].maxminute := 16, [111].log_data[42].valid := 1, [111].log_data[43].min := -0.27999878, [111].log_data[43].max := -0.26000214, [111].log_data[43].total := -936.7883, [111].log_data[43].time := 3600.0, [111].log_data[43].valid := 1, [111].log_data[44].min := -0.30000305, [111].log_data[44].max := -0.27999878, [111].log_data[44].total := -1080.081, [111].log_data[44].time := 3600.0, [111].log_data[44].maxminute := 12, [111].log_data[44].valid := 1, [111].log_data[45].time := 3600.0, [111].log_data[45].valid := 1, [111].log_data[46].time := 3600.0, [111].log_data[46].valid := 1, [111].log_data[47].time := 3600.0, [111].log_data[47].valid := 1, [111].log_data[48].min := 6.5708866, [111].log_data[48].max := 6.903678, [111].log_data[48].total := 24173.697, [111].log_data[48].time := 3600.0, [111].log_data[48].minminute := 42, [111].log_data[48].maxminute := 22, [111].log_data[48].valid := 1, [111].log_data[49].min := 6.5920205, [111].log_data[49].max := 9.460231, [111].log_data[49].total := 28765.398, [111].log_data[49].time := 3600.0, [111].log_data[49].minminute := 42, [111].log_data[49].maxminute := 14, [111].log_data[49].valid := 1, [111].log_data[50].min := 1.8143013, [111].log_data[50].max := 1.9200629, [111].log_data[50].total := 6756.339, [111].log_data[50].time := 3600.0, [111].log_data[50].minminute := 15,
        [111].log_data[50].maxminute := 24, [111].log_data[50].valid := 1, [111].log_data[51].time := 3600.0, [111].log_data[51].valid := 1, [111].log_data[52].min := -3.0200043, [111].log_data[52].max := 0.11999512, [111].log_data[52].total := -7997.063, [111].log_data[52].time := 3600.0, [111].log_data[52].minminute := 19, [111].log_data[52].maxminute := 7, [111].log_data[52].valid := 1, [111].log_data[53].min := -2.5200043, [111].log_data[53].max := 0.17999268, [111].log_data[53].total := -7368.0913, [111].log_data[53].time := 3600.0, [111].log_data[53].minminute := 11, [111].log_data[53].maxminute := 24, [111].log_data[53].valid := 1, [111].log_data[54].max := 0.557, [111].log_data[54].total := 1254.7563, [111].log_data[54].time := 3600.0, [111].log_data[54].minminute := 7, [111].log_data[54].maxminute := 19, [111].log_data[54].valid := 1, [111].log_data[55].max := 0.5335, [111].log_data[55].total := 1217.2458, [111].log_data[55].time := 3600.0, [111].log_data[55].minminute := 2, [111].log_data[55].maxminute := 25, [111].log_data[55].valid := 1, [111].log_data[56].min := 0.15930341, [111].log_data[56].max := 0.15985303, [111].log_data[56].total := 574.358, [111].log_data[56].time := 3600.0, [111].log_data[56].minminute := 15, [111].log_data[56].maxminute := 6, [111].log_data[56].valid := 1, [111].log_data[57].min := 0.2229018, [111].log_data[57].max := 0.22521807, [111].log_data[57].total := 808.2129, [111].log_data[57].time := 3600.0, [111].log_data[57].minminute := 51, [111].log_data[57].valid := 1, [111].log_data[58].time := 3600.0, [111].log_data[58].valid := 1, [111].log_data[59].time := 3600.0, [111].log_data[59].valid := 1, [111].log_data[60].valid := 1, [111].log_data[61].valid := 1, [111].log_data[62].valid := 1, [111].log_data[63].valid := 1, [111].log_data[64].valid := 1, [111].log_data[65].valid := 1, [111].log_data[66].valid := 1, [111].log_data[67].valid := 1, [111].log_data[68].valid := 1, [111].log_data[69].valid := 1, [111].log_data[70].valid := 1, [111].log_data[71].valid := 1, [111].log_data[72].valid := 1,
        [111].log_data[73].valid := 1, [111].log_data[74].valid := 1, [111].log_data[75].valid := 1, [111].log_data[76].valid := 1, [111].log_data[77].valid := 1, [111].log_data[78].valid := 1, [111].log_data[79].valid := 1, [111].log_data[80].valid := 1, [111].log_data[81].valid := 1, [111].log_data[82].valid := 1, [111].log_data[83].valid := 1, [111].log_data[84].valid := 1, [111].log_data[85].valid := 1, [111].log_data[86].valid := 1, [111].log_data[87].valid := 1, [111].log_data[88].valid := 1, [111].log_data[89].valid := 1, [111].log_data[90].valid := 1, [111].log_data[91].valid := 1, [111].log_data[92].valid := 1, [111].log_data[93].valid := 1, [111].log_data[94].valid := 1, [111].log_data[95].valid := 1, [111].log_data[96].valid := 1, [111].log_data[97].valid := 1, [111].log_data[98].valid := 1, [111].log_data[99].valid := 1, [111].log_data[100].valid := 1, [111].log_data[101].valid := 1, [111].log_data[102].valid := 1, [111].log_data[103].valid := 1, [111].log_data[104].valid := 1, [111].log_data[105].valid := 1, [111].log_data[106].valid := 1, [111].log_data[107].valid := 1, [111].log_data[108].valid := 1, [111].log_data[109].valid := 1, [111].log_data[110].valid := 1, [111].log_data[111].valid := 1, [111].log_data[112].valid := 1, [111].log_data[113].valid := 1, [111].log_data[114].valid := 1, [111].log_data[115].valid := 1, [111].log_data[116].valid := 1, [111].log_data[117].valid := 1, [111].log_data[118].valid := 1, [111].log_data[119].valid := 1, [111].log_data[120].valid := 1, [111].log_data[121].valid := 1, [111].log_data[122].valid := 1, [111].log_data[123].valid := 1, [111].log_data[124].valid := 1, [111].time.Year := 2023, [111].time.Month := 1, [111].time.Day := 17, [111].time.Hour := 18, [111].time.Minute := 59, [111].time.Second := 59, [112].log_data[0].min := 1.0, [112].log_data[0].max := 1.0,
        [112].log_data[0].total := 3600.0, [112].log_data[0].time := 3600.0, [112].log_data[0].valid := 1, [112].log_data[1].max := 1.0, [112].log_data[1].total := 549.5, [112].log_data[1].time := 3600.0, [112].log_data[1].maxminute := 31, [112].log_data[1].valid := 1, [112].log_data[2].max := 1.0, [112].log_data[2].total := 546.0, [112].log_data[2].time := 3600.0, [112].log_data[2].maxminute := 31, [112].log_data[2].valid := 1, [112].log_data[3].time := 3600.0, [112].log_data[3].valid := 1, [112].log_data[4].time := 3600.0, [112].log_data[4].valid := 1, [112].log_data[5].max := 1.0, [112].log_data[5].total := 247.5, [112].log_data[5].time := 3600.0, [112].log_data[5].maxminute := 33, [112].log_data[5].valid := 1, [112].log_data[6].time := 3600.0, [112].log_data[6].valid := 1, [112].log_data[7].time := 3600.0, [112].log_data[7].valid := 1, [112].log_data[8].min := 1.0, [112].log_data[8].max := 1.0, [112].log_data[8].total := 3600.0, [112].log_data[8].time := 3600.0, [112].log_data[8].valid := 1, [112].log_data[9].min := 1.0, [112].log_data[9].max := 1.0, [112].log_data[9].total := 3600.0, [112].log_data[9].time := 3600.0, [112].log_data[9].valid := 1, [112].log_data[10].min := 1.0, [112].log_data[10].max := 1.0, [112].log_data[10].total := 3600.0, [112].log_data[10].time := 3600.0, [112].log_data[10].valid := 1, [112].log_data[11].time := 3600.0, [112].log_data[11].valid := 1, [112].log_data[12].min := 1.0, [112].log_data[12].max := 1.0, [112].log_data[12].total := 3600.0, [112].log_data[12].time := 3600.0, [112].log_data[12].valid := 1, [112].log_data[13].min := 1.0, [112].log_data[13].max := 1.0, [112].log_data[13].total := 3600.0, [112].log_data[13].time := 3600.0, [112].log_data[13].valid := 1, [112].log_data[14].time := 3600.0, [112].log_data[14].valid := 1, [112].log_data[15].time := 3600.0, [112].log_data[15].valid := 1, [112].log_data[16].time := 3600.0, [112].log_data[16].valid := 1, [112].log_data[17].min := 1.0,
        [112].log_data[17].max := 1.0, [112].log_data[17].total := 3600.0, [112].log_data[17].time := 3600.0, [112].log_data[17].valid := 1, [112].log_data[18].time := 3600.0, [112].log_data[18].valid := 1, [112].log_data[19].time := 3600.0, [112].log_data[19].valid := 1, [112].log_data[20].time := 3600.0, [112].log_data[20].valid := 1, [112].log_data[21].min := 1.0, [112].log_data[21].max := 1.0, [112].log_data[21].total := 3600.0, [112].log_data[21].time := 3600.0, [112].log_data[21].valid := 1, [112].log_data[22].time := 3600.0, [112].log_data[22].valid := 1, [112].log_data[23].time := 3600.0, [112].log_data[23].valid := 1, [112].log_data[24].time := 3600.0, [112].log_data[24].valid := 1, [112].log_data[25].time := 3600.0, [112].log_data[25].valid := 1, [112].log_data[26].time := 3600.0, [112].log_data[26].valid := 1, [112].log_data[27].time := 3600.0, [112].log_data[27].valid := 1, [112].log_data[28].time := 3600.0, [112].log_data[28].valid := 1, [112].log_data[29].min := 1.0, [112].log_data[29].max := 1.0, [112].log_data[29].total := 3600.0, [112].log_data[29].time := 3600.0, [112].log_data[29].valid := 1, [112].log_data[30].min := 1.0, [112].log_data[30].max := 1.0, [112].log_data[30].total := 3600.0, [112].log_data[30].time := 3600.0, [112].log_data[30].valid := 1, [112].log_data[31].max := 1.0, [112].log_data[31].total := 1629.749, [112].log_data[31].time := 3600.0, [112].log_data[31].maxminute := 1, [112].log_data[31].valid := 1, [112].log_data[32].max := 1.0, [112].log_data[32].total := 1440.2471, [112].log_data[32].time := 3600.0, [112].log_data[32].valid := 1, [112].log_data[33].time := 3600.0, [112].log_data[33].valid := 1, [112].log_data[34].time := 3600.0, [112].log_data[34].valid := 1, [112].log_data[35].max := 1.0, [112].log_data[35].total := 1440.7471, [112].log_data[35].time := 3600.0, [112].log_data[35].minminute := 5, [112].log_data[35].valid := 1, [112].log_data[36].max := 1.0, [112].log_data[36].total := 1629.7471, [112].log_data[36].time := 3600.0,
        [112].log_data[36].maxminute := 7, [112].log_data[36].valid := 1, [112].log_data[37].max := 7.6050467, [112].log_data[37].total := 3628.5386, [112].log_data[37].time := 3600.0, [112].log_data[37].maxminute := 33, [112].log_data[37].valid := 1, [112].log_data[38].time := 3600.0, [112].log_data[38].valid := 1, [112].log_data[39].min := 0.99529505, [112].log_data[39].max := 1.0216767, [112].log_data[39].total := 3606.9604, [112].log_data[39].time := 3600.0, [112].log_data[39].minminute := 47, [112].log_data[39].maxminute := 38, [112].log_data[39].valid := 1, [112].log_data[40].min := 7.5843773, [112].log_data[40].max := 7.6162558, [112].log_data[40].total := 27364.926, [112].log_data[40].time := 3600.0, [112].log_data[40].minminute := 17, [112].log_data[40].maxminute := 21, [112].log_data[40].valid := 1, [112].log_data[41].min := 0.02273633, [112].log_data[41].max := 0.023325196, [112].log_data[41].total := 82.60551, [112].log_data[41].time := 3600.0, [112].log_data[41].maxminute := 34, [112].log_data[41].valid := 1, [112].log_data[42].min := 2.291407, [112].log_data[42].max := 2.296118, [112].log_data[42].total := 8258.973, [112].log_data[42].time := 3600.0, [112].log_data[42].minminute := 13, [112].log_data[42].maxminute := 31, [112].log_data[42].valid := 1, [112].log_data[43].min := -0.27999878, [112].log_data[43].max := -0.26000214, [112].log_data[43].total := -938.2508, [112].log_data[43].time := 3600.0, [112].log_data[43].minminute := 2, [112].log_data[43].valid := 1, [112].log_data[44].min := -0.30000305, [112].log_data[44].max := -0.27999878, [112].log_data[44].total := -1080.086, [112].log_data[44].time := 3600.0, [112].log_data[44].maxminute := 28, [112].log_data[44].valid := 1, [112].log_data[45].time := 3600.0, [112].log_data[45].valid := 1, [112].log_data[46].time := 3600.0, [112].log_data[46].valid := 1, [112].log_data[47].time := 3600.0, [112].log_data[47].valid := 1, [112].log_data[48].min := 6.585176, [112].log_data[48].max := 6.893785, [112].log_data[48].total := 24279.049, [112].log_data[48].time := 3600.0, [112].log_data[48].minminute := 59, [112].log_data[48].maxminute := 40,
